Fanuc TP program (LS listing): qwerty_12.ls

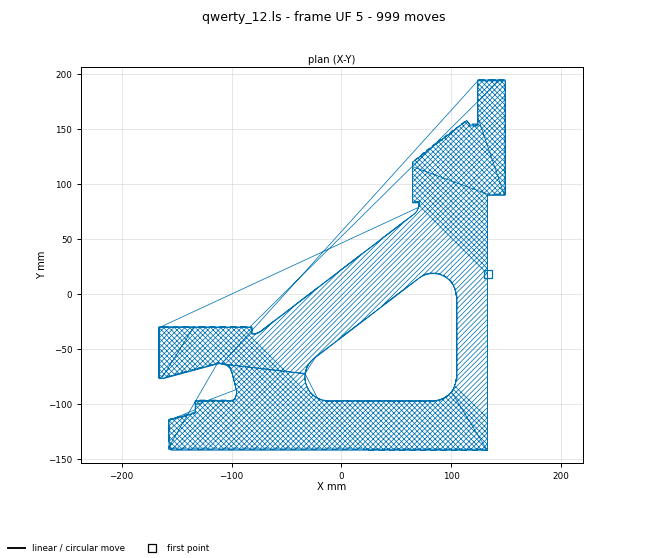
[picture p0: tool path of qwerty_12.ls in frame UF 5, 999 of 999 moves have a stored position in this frame; points joined in program order, loops and branches not executed]
/PROG qwerty_12
/ATTR
OWNER       = MNEDITOR;
CREATE      = DATE 100-11-20  TIME 09:43:21;
MODIFIED    = DATE 100-12-05  TIME 05:26:29;
LINE_COUNT = 999;
PROTECT     = READ_WRITE;
TCD:  STACK_SIZE    = 0,
      TASK_PRIORITY = 50,
      TIME_SLICE    = 0,
      BUSY_LAMP_OFF = 0,
      ABORT_REQUEST = 0,
      PAUSE_REQUEST = 0;
DEFAULT_GROUP   = 1,1,*,*,*;
CONTROL_CODE    = 00000000 00000000;
/MN
1: L P[1] WELD_SPEED CNT100 COORD PTH  ;
2: L P[2] WELD_SPEED CNT100 COORD PTH  ;
3: L P[3] WELD_SPEED CNT100 COORD PTH  ;
4: L P[4] WELD_SPEED CNT100 COORD PTH  ;
5: L P[5] WELD_SPEED CNT100 COORD PTH  ;
6: L P[6] WELD_SPEED CNT100 COORD PTH  ;
7: L P[7] WELD_SPEED CNT100 COORD PTH  ;
8: L P[8] WELD_SPEED CNT100 COORD PTH  ;
9: L P[9] WELD_SPEED CNT100 COORD PTH  ;
10: L P[10] WELD_SPEED CNT100 COORD PTH  ;
11: L P[11] WELD_SPEED CNT100 COORD PTH  ;
12: L P[12] WELD_SPEED CNT100 COORD PTH  ;
13: L P[13] WELD_SPEED CNT100 COORD PTH  ;
14: L P[14] WELD_SPEED CNT100 COORD PTH  ;
15: L P[15] WELD_SPEED CNT100 COORD PTH  ;
16: L P[16] WELD_SPEED CNT100 COORD PTH  ;
17: L P[17] WELD_SPEED CNT100 COORD PTH  ;
18: L P[18] WELD_SPEED CNT100 COORD PTH  ;
19: L P[19] WELD_SPEED CNT100 COORD PTH  ;
20: L P[20] WELD_SPEED CNT100 COORD PTH  ;
21: L P[21] WELD_SPEED CNT100 COORD PTH  ;
22: L P[22] WELD_SPEED CNT100 COORD PTH  ;
23: L P[23] WELD_SPEED CNT100 COORD PTH  ;
24: L P[24] WELD_SPEED CNT100 COORD PTH  ;
25: L P[25] WELD_SPEED CNT100 COORD PTH  ;
26: L P[26] WELD_SPEED CNT100 COORD PTH  ;
27: L P[27] WELD_SPEED CNT100 COORD PTH  ;
28: L P[28] WELD_SPEED CNT100 COORD PTH  ;
29: L P[29] WELD_SPEED CNT100 COORD PTH  ;
30: L P[30] WELD_SPEED CNT100 COORD PTH  ;
31: L P[31] WELD_SPEED CNT100 COORD PTH  ;
32: L P[32] WELD_SPEED CNT100 COORD PTH  ;
33: L P[33] WELD_SPEED CNT100 COORD PTH  ;
34: L P[34] WELD_SPEED CNT100 COORD PTH  ;
35: L P[35] WELD_SPEED CNT100 COORD PTH  ;
36: L P[36] WELD_SPEED CNT100 COORD PTH  ;
37: L P[37] WELD_SPEED CNT100 COORD PTH  ;
38: L P[38] WELD_SPEED CNT100 COORD PTH  ;
39: L P[39] WELD_SPEED CNT100 COORD PTH  ;
40: L P[40] WELD_SPEED CNT100 COORD PTH  ;
41: L P[41] WELD_SPEED CNT100 COORD PTH  ;
42: L P[42] WELD_SPEED CNT100 COORD PTH  ;
43: L P[43] WELD_SPEED CNT100 COORD PTH  ;
44: L P[44] WELD_SPEED CNT100 COORD PTH  ;
45: L P[45] WELD_SPEED CNT100 COORD PTH  ;
46: L P[46] WELD_SPEED CNT100 COORD PTH  ;
47: L P[47] WELD_SPEED CNT100 COORD PTH  ;
48: L P[48] WELD_SPEED CNT100 COORD PTH  ;
49: L P[49] WELD_SPEED CNT100 COORD PTH  ;
50: L P[50] WELD_SPEED CNT100 COORD PTH  ;
51: L P[51] WELD_SPEED CNT100 COORD PTH  ;
52: L P[52] WELD_SPEED CNT100 COORD PTH  ;
53: L P[53] WELD_SPEED CNT100 COORD PTH  ;
54: L P[54] WELD_SPEED CNT100 COORD PTH  ;
55: L P[55] WELD_SPEED CNT100 COORD PTH  ;
56: L P[56] WELD_SPEED CNT100 COORD PTH  ;
57: L P[57] WELD_SPEED CNT100 COORD PTH  ;
58: L P[58] WELD_SPEED CNT100 COORD PTH  ;
59: L P[59] WELD_SPEED CNT100 COORD PTH  ;
60: L P[60] WELD_SPEED CNT100 COORD PTH  ;
61: L P[61] WELD_SPEED CNT100 COORD PTH  ;
62: L P[62] WELD_SPEED CNT100 COORD PTH  ;
63: L P[63] WELD_SPEED CNT100 COORD PTH  ;
64: L P[64] WELD_SPEED CNT100 COORD PTH  ;
65: L P[65] WELD_SPEED CNT100 COORD PTH  ;
66: L P[66] WELD_SPEED CNT100 COORD PTH  ;
67: L P[67] WELD_SPEED CNT100 COORD PTH  ;
68: L P[68] WELD_SPEED CNT100 COORD PTH  ;
69: L P[69] WELD_SPEED CNT100 COORD PTH  ;
70: L P[70] WELD_SPEED CNT100 COORD PTH  ;
71: L P[71] WELD_SPEED CNT100 COORD PTH  ;
72: L P[72] WELD_SPEED CNT100 COORD PTH  ;
73: L P[73] WELD_SPEED CNT100 COORD PTH  ;
74: L P[74] WELD_SPEED CNT100 COORD PTH  ;
75: L P[75] WELD_SPEED CNT100 COORD PTH  ;
76: L P[76] WELD_SPEED CNT100 COORD PTH  ;
77: L P[77] WELD_SPEED CNT100 COORD PTH  ;
78: L P[78] WELD_SPEED CNT100 COORD PTH  ;
79: L P[79] WELD_SPEED CNT100 COORD PTH  ;
80: L P[80] WELD_SPEED CNT100 COORD PTH  ;
81: L P[81] WELD_SPEED CNT100 COORD PTH  ;
82: L P[82] WELD_SPEED CNT100 COORD PTH  ;
83: L P[83] WELD_SPEED CNT100 COORD PTH  ;
84: L P[84] WELD_SPEED CNT100 COORD PTH  ;
85: L P[85] WELD_SPEED CNT100 COORD PTH  ;
86: L P[86] WELD_SPEED CNT100 COORD PTH  ;
87: L P[87] WELD_SPEED CNT100 COORD PTH  ;
88: L P[88] WELD_SPEED CNT100 COORD PTH  ;
: Arc End[1];
89: L P[89] 240cm/min CNT100 COORD  ;
: Arc Start[1];
90: L P[90] WELD_SPEED CNT100 COORD PTH  ;
91: L P[91] WELD_SPEED CNT100 COORD PTH  ;
92: L P[92] WELD_SPEED CNT100 COORD PTH  ;
93: L P[93] WELD_SPEED CNT100 COORD PTH  ;
94: L P[94] WELD_SPEED CNT100 COORD PTH  ;
95: L P[95] WELD_SPEED CNT100 COORD PTH  ;
96: L P[96] WELD_SPEED CNT100 COORD PTH  ;
97: L P[97] WELD_SPEED CNT100 COORD PTH  ;
98: L P[98] WELD_SPEED CNT100 COORD PTH  ;
99: L P[99] WELD_SPEED CNT100 COORD PTH  ;
100: L P[100] WELD_SPEED CNT100 COORD PTH  ;
101: L P[101] WELD_SPEED CNT100 COORD PTH  ;
102: L P[102] WELD_SPEED CNT100 COORD PTH  ;
103: L P[103] WELD_SPEED CNT100 COORD PTH  ;
104: L P[104] WELD_SPEED CNT100 COORD PTH  ;
105: L P[105] WELD_SPEED CNT100 COORD PTH  ;
106: L P[106] WELD_SPEED CNT100 COORD PTH  ;
107: L P[107] WELD_SPEED CNT100 COORD PTH  ;
108: L P[108] WELD_SPEED CNT100 COORD PTH  ;
109: L P[109] WELD_SPEED CNT100 COORD PTH  ;
110: L P[110] WELD_SPEED CNT100 COORD PTH  ;
111: L P[111] WELD_SPEED CNT100 COORD PTH  ;
112: L P[112] WELD_SPEED CNT100 COORD PTH  ;
: Arc End[1];
113: L P[113] 240cm/min CNT100 COORD  ;
: Arc Start[1];
114: L P[114] WELD_SPEED CNT100 COORD PTH  ;
115: L P[115] WELD_SPEED CNT100 COORD PTH  ;
116: L P[116] WELD_SPEED CNT100 COORD PTH  ;
117: L P[117] WELD_SPEED CNT100 COORD PTH  ;
118: L P[118] WELD_SPEED CNT100 COORD PTH  ;
119: L P[119] WELD_SPEED CNT100 COORD PTH  ;
120: L P[120] WELD_SPEED CNT100 COORD PTH  ;
121: L P[121] WELD_SPEED CNT100 COORD PTH  ;
122: L P[122] WELD_SPEED CNT100 COORD PTH  ;
123: L P[123] WELD_SPEED CNT100 COORD PTH  ;
124: L P[124] WELD_SPEED CNT100 COORD PTH  ;
125: L P[125] WELD_SPEED CNT100 COORD PTH  ;
126: L P[126] WELD_SPEED CNT100 COORD PTH  ;
127: L P[127] WELD_SPEED CNT100 COORD PTH  ;
128: L P[128] WELD_SPEED CNT100 COORD PTH  ;
129: L P[129] WELD_SPEED CNT100 COORD PTH  ;
130: L P[130] WELD_SPEED CNT100 COORD PTH  ;
131: L P[131] WELD_SPEED CNT100 COORD PTH  ;
132: L P[132] WELD_SPEED CNT100 COORD PTH  ;
133: L P[133] WELD_SPEED CNT100 COORD PTH  ;
134: L P[134] WELD_SPEED CNT100 COORD PTH  ;
135: L P[135] WELD_SPEED CNT100 COORD PTH  ;
136: L P[136] WELD_SPEED CNT100 COORD PTH  ;
137: L P[137] WELD_SPEED CNT100 COORD PTH  ;
138: L P[138] WELD_SPEED CNT100 COORD PTH  ;
139: L P[139] WELD_SPEED CNT100 COORD PTH  ;
140: L P[140] WELD_SPEED CNT100 COORD PTH  ;
141: L P[141] WELD_SPEED CNT100 COORD PTH  ;
142: L P[142] WELD_SPEED CNT100 COORD PTH  ;
143: L P[143] WELD_SPEED CNT100 COORD PTH  ;
144: L P[144] WELD_SPEED CNT100 COORD PTH  ;
145: L P[145] WELD_SPEED CNT100 COORD PTH  ;
146: L P[146] WELD_SPEED CNT100 COORD PTH  ;
147: L P[147] WELD_SPEED CNT100 COORD PTH  ;
148: L P[148] WELD_SPEED CNT100 COORD PTH  ;
149: L P[149] WELD_SPEED CNT100 COORD PTH  ;
150: L P[150] WELD_SPEED CNT100 COORD PTH  ;
151: L P[151] WELD_SPEED CNT100 COORD PTH  ;
152: L P[152] WELD_SPEED CNT100 COORD PTH  ;
153: L P[153] WELD_SPEED CNT100 COORD PTH  ;
154: L P[154] WELD_SPEED CNT100 COORD PTH  ;
155: L P[155] WELD_SPEED CNT100 COORD PTH  ;
156: L P[156] WELD_SPEED CNT100 COORD PTH  ;
157: L P[157] WELD_SPEED CNT100 COORD PTH  ;
158: L P[158] WELD_SPEED CNT100 COORD PTH  ;
159: L P[159] WELD_SPEED CNT100 COORD PTH  ;
160: L P[160] WELD_SPEED CNT100 COORD PTH  ;
161: L P[161] WELD_SPEED CNT100 COORD PTH  ;
162: L P[162] WELD_SPEED CNT100 COORD PTH  ;
163: L P[163] WELD_SPEED CNT100 COORD PTH  ;
164: L P[164] WELD_SPEED CNT100 COORD PTH  ;
165: L P[165] WELD_SPEED CNT100 COORD PTH  ;
166: L P[166] WELD_SPEED CNT100 COORD PTH  ;
167: L P[167] WELD_SPEED CNT100 COORD PTH  ;
168: L P[168] WELD_SPEED CNT100 COORD PTH  ;
169: L P[169] WELD_SPEED CNT100 COORD PTH  ;
170: L P[170] WELD_SPEED CNT100 COORD PTH  ;
171: L P[171] WELD_SPEED CNT100 COORD PTH  ;
172: L P[172] WELD_SPEED CNT100 COORD PTH  ;
173: L P[173] WELD_SPEED CNT100 COORD PTH  ;
174: L P[174] WELD_SPEED CNT100 COORD PTH  ;
175: L P[175] WELD_SPEED CNT100 COORD PTH  ;
176: L P[176] WELD_SPEED CNT100 COORD PTH  ;
177: L P[177] WELD_SPEED CNT100 COORD PTH  ;
178: L P[178] WELD_SPEED CNT100 COORD PTH  ;
179: L P[179] WELD_SPEED CNT100 COORD PTH  ;
180: L P[180] WELD_SPEED CNT100 COORD PTH  ;
181: L P[181] WELD_SPEED CNT100 COORD PTH  ;
182: L P[182] WELD_SPEED CNT100 COORD PTH  ;
183: L P[183] WELD_SPEED CNT100 COORD PTH  ;
184: L P[184] WELD_SPEED CNT100 COORD PTH  ;
185: L P[185] WELD_SPEED CNT100 COORD PTH  ;
186: L P[186] WELD_SPEED CNT100 COORD PTH  ;
187: L P[187] WELD_SPEED CNT100 COORD PTH  ;
188: L P[188] WELD_SPEED CNT100 COORD PTH  ;
189: L P[189] WELD_SPEED CNT100 COORD PTH  ;
190: L P[190] WELD_SPEED CNT100 COORD PTH  ;
191: L P[191] WELD_SPEED CNT100 COORD PTH  ;
192: L P[192] WELD_SPEED CNT100 COORD PTH  ;
193: L P[193] WELD_SPEED CNT100 COORD PTH  ;
194: L P[194] WELD_SPEED CNT100 COORD PTH  ;
195: L P[195] WELD_SPEED CNT100 COORD PTH  ;
196: L P[196] WELD_SPEED CNT100 COORD PTH  ;
197: L P[197] WELD_SPEED CNT100 COORD PTH  ;
198: L P[198] WELD_SPEED CNT100 COORD PTH  ;
199: L P[199] WELD_SPEED CNT100 COORD PTH  ;
200: L P[200] WELD_SPEED CNT100 COORD PTH  ;
201: L P[201] WELD_SPEED CNT100 COORD PTH  ;
202: L P[202] WELD_SPEED CNT100 COORD PTH  ;
203: L P[203] WELD_SPEED CNT100 COORD PTH  ;
204: L P[204] WELD_SPEED CNT100 COORD PTH  ;
205: L P[205] WELD_SPEED CNT100 COORD PTH  ;
206: L P[206] WELD_SPEED CNT100 COORD PTH  ;
207: L P[207] WELD_SPEED CNT100 COORD PTH  ;
208: L P[208] WELD_SPEED CNT100 COORD PTH  ;
209: L P[209] WELD_SPEED CNT100 COORD PTH  ;
210: L P[210] WELD_SPEED CNT100 COORD PTH  ;
211: L P[211] WELD_SPEED CNT100 COORD PTH  ;
212: L P[212] WELD_SPEED CNT100 COORD PTH  ;
213: L P[213] WELD_SPEED CNT100 COORD PTH  ;
214: L P[214] WELD_SPEED CNT100 COORD PTH  ;
215: L P[215] WELD_SPEED CNT100 COORD PTH  ;
: Arc End[1];
216: L P[216] 240cm/min CNT100 COORD  ;
217: L P[217] 240cm/min CNT100 COORD  ;
: Arc Start[1];
218: L P[218] WELD_SPEED CNT100 COORD PTH  ;
219: L P[219] WELD_SPEED CNT100 COORD PTH  ;
220: L P[220] WELD_SPEED CNT100 COORD PTH  ;
221: L P[221] WELD_SPEED CNT100 COORD PTH  ;
222: L P[222] WELD_SPEED CNT100 COORD PTH  ;
223: L P[223] WELD_SPEED CNT100 COORD PTH  ;
224: L P[224] WELD_SPEED CNT100 COORD PTH  ;
225: L P[225] WELD_SPEED CNT100 COORD PTH  ;
226: L P[226] WELD_SPEED CNT100 COORD PTH  ;
227: L P[227] WELD_SPEED CNT100 COORD PTH  ;
228: L P[228] WELD_SPEED CNT100 COORD PTH  ;
229: L P[229] WELD_SPEED CNT100 COORD PTH  ;
230: L P[230] WELD_SPEED CNT100 COORD PTH  ;
231: L P[231] WELD_SPEED CNT100 COORD PTH  ;
232: L P[232] WELD_SPEED CNT100 COORD PTH  ;
233: L P[233] WELD_SPEED CNT100 COORD PTH  ;
234: L P[234] WELD_SPEED CNT100 COORD PTH  ;
235: L P[235] WELD_SPEED CNT100 COORD PTH  ;
236: L P[236] WELD_SPEED CNT100 COORD PTH  ;
237: L P[237] WELD_SPEED CNT100 COORD PTH  ;
238: L P[238] WELD_SPEED CNT100 COORD PTH  ;
239: L P[239] WELD_SPEED CNT100 COORD PTH  ;
240: L P[240] WELD_SPEED CNT100 COORD PTH  ;
241: L P[241] WELD_SPEED CNT100 COORD PTH  ;
242: L P[242] WELD_SPEED CNT100 COORD PTH  ;
243: L P[243] WELD_SPEED CNT100 COORD PTH  ;
244: L P[244] WELD_SPEED CNT100 COORD PTH  ;
245: L P[245] WELD_SPEED CNT100 COORD PTH  ;
246: L P[246] WELD_SPEED CNT100 COORD PTH  ;
247: L P[247] WELD_SPEED CNT100 COORD PTH  ;
248: L P[248] WELD_SPEED CNT100 COORD PTH  ;
249: L P[249] WELD_SPEED CNT100 COORD PTH  ;
250: L P[250] WELD_SPEED CNT100 COORD PTH  ;
251: L P[251] WELD_SPEED CNT100 COORD PTH  ;
252: L P[252] WELD_SPEED CNT100 COORD PTH  ;
253: L P[253] WELD_SPEED CNT100 COORD PTH  ;
254: L P[254] WELD_SPEED CNT100 COORD PTH  ;
255: L P[255] WELD_SPEED CNT100 COORD PTH  ;
256: L P[256] WELD_SPEED CNT100 COORD PTH  ;
257: L P[257] WELD_SPEED CNT100 COORD PTH  ;
258: L P[258] WELD_SPEED CNT100 COORD PTH  ;
259: L P[259] WELD_SPEED CNT100 COORD PTH  ;
260: L P[260] WELD_SPEED CNT100 COORD PTH  ;
261: L P[261] WELD_SPEED CNT100 COORD PTH  ;
262: L P[262] WELD_SPEED CNT100 COORD PTH  ;
263: L P[263] WELD_SPEED CNT100 COORD PTH  ;
264: L P[264] WELD_SPEED CNT100 COORD PTH  ;
265: L P[265] WELD_SPEED CNT100 COORD PTH  ;
266: L P[266] WELD_SPEED CNT100 COORD PTH  ;
267: L P[267] WELD_SPEED CNT100 COORD PTH  ;
268: L P[268] WELD_SPEED CNT100 COORD PTH  ;
269: L P[269] WELD_SPEED CNT100 COORD PTH  ;
270: L P[270] WELD_SPEED CNT100 COORD PTH  ;
271: L P[271] WELD_SPEED CNT100 COORD PTH  ;
272: L P[272] WELD_SPEED CNT100 COORD PTH  ;
273: L P[273] WELD_SPEED CNT100 COORD PTH  ;
274: L P[274] WELD_SPEED CNT100 COORD PTH  ;
275: L P[275] WELD_SPEED CNT100 COORD PTH  ;
276: L P[276] WELD_SPEED CNT100 COORD PTH  ;
: Arc End[1];
277: L P[277] 240cm/min CNT100 COORD  ;
: Arc Start[1];
278: L P[278] WELD_SPEED CNT100 COORD PTH  ;
279: L P[279] WELD_SPEED CNT100 COORD PTH  ;
280: L P[280] WELD_SPEED CNT100 COORD PTH  ;
281: L P[281] WELD_SPEED CNT100 COORD PTH  ;
282: L P[282] WELD_SPEED CNT100 COORD PTH  ;
283: L P[283] WELD_SPEED CNT100 COORD PTH  ;
284: L P[284] WELD_SPEED CNT100 COORD PTH  ;
285: L P[285] WELD_SPEED CNT100 COORD PTH  ;
286: L P[286] WELD_SPEED CNT100 COORD PTH  ;
287: L P[287] WELD_SPEED CNT100 COORD PTH  ;
288: L P[288] WELD_SPEED CNT100 COORD PTH  ;
289: L P[289] WELD_SPEED CNT100 COORD PTH  ;
290: L P[290] WELD_SPEED CNT100 COORD PTH  ;
291: L P[291] WELD_SPEED CNT100 COORD PTH  ;
292: L P[292] WELD_SPEED CNT100 COORD PTH  ;
293: L P[293] WELD_SPEED CNT100 COORD PTH  ;
294: L P[294] WELD_SPEED CNT100 COORD PTH  ;
295: L P[295] WELD_SPEED CNT100 COORD PTH  ;
296: L P[296] WELD_SPEED CNT100 COORD PTH  ;
297: L P[297] WELD_SPEED CNT100 COORD PTH  ;
298: L P[298] WELD_SPEED CNT100 COORD PTH  ;
299: L P[299] WELD_SPEED CNT100 COORD PTH  ;
300: L P[300] WELD_SPEED CNT100 COORD PTH  ;
301: L P[301] WELD_SPEED CNT100 COORD PTH  ;
302: L P[302] WELD_SPEED CNT100 COORD PTH  ;
303: L P[303] WELD_SPEED CNT100 COORD PTH  ;
304: L P[304] WELD_SPEED CNT100 COORD PTH  ;
305: L P[305] WELD_SPEED CNT100 COORD PTH  ;
306: L P[306] WELD_SPEED CNT100 COORD PTH  ;
307: L P[307] WELD_SPEED CNT100 COORD PTH  ;
308: L P[308] WELD_SPEED CNT100 COORD PTH  ;
309: L P[309] WELD_SPEED CNT100 COORD PTH  ;
310: L P[310] WELD_SPEED CNT100 COORD PTH  ;
311: L P[311] WELD_SPEED CNT100 COORD PTH  ;
312: L P[312] WELD_SPEED CNT100 COORD PTH  ;
313: L P[313] WELD_SPEED CNT100 COORD PTH  ;
314: L P[314] WELD_SPEED CNT100 COORD PTH  ;
315: L P[315] WELD_SPEED CNT100 COORD PTH  ;
316: L P[316] WELD_SPEED CNT100 COORD PTH  ;
317: L P[317] WELD_SPEED CNT100 COORD PTH  ;
318: L P[318] WELD_SPEED CNT100 COORD PTH  ;
319: L P[319] WELD_SPEED CNT100 COORD PTH  ;
320: L P[320] WELD_SPEED CNT100 COORD PTH  ;
321: L P[321] WELD_SPEED CNT100 COORD PTH  ;
322: L P[322] WELD_SPEED CNT100 COORD PTH  ;
323: L P[323] WELD_SPEED CNT100 COORD PTH  ;
324: L P[324] WELD_SPEED CNT100 COORD PTH  ;
325: L P[325] WELD_SPEED CNT100 COORD PTH  ;
326: L P[326] WELD_SPEED CNT100 COORD PTH  ;
327: L P[327] WELD_SPEED CNT100 COORD PTH  ;
328: L P[328] WELD_SPEED CNT100 COORD PTH  ;
329: L P[329] WELD_SPEED CNT100 COORD PTH  ;
330: L P[330] WELD_SPEED CNT100 COORD PTH  ;
331: L P[331] WELD_SPEED CNT100 COORD PTH  ;
332: L P[332] WELD_SPEED CNT100 COORD PTH  ;
333: L P[333] WELD_SPEED CNT100 COORD PTH  ;
334: L P[334] WELD_SPEED CNT100 COORD PTH  ;
335: L P[335] WELD_SPEED CNT100 COORD PTH  ;
336: L P[336] WELD_SPEED CNT100 COORD PTH  ;
337: L P[337] WELD_SPEED CNT100 COORD PTH  ;
338: L P[338] WELD_SPEED CNT100 COORD PTH  ;
339: L P[339] WELD_SPEED CNT100 COORD PTH  ;
340: L P[340] WELD_SPEED CNT100 COORD PTH  ;
341: L P[341] WELD_SPEED CNT100 COORD PTH  ;
342: L P[342] WELD_SPEED CNT100 COORD PTH  ;
343: L P[343] WELD_SPEED CNT100 COORD PTH  ;
344: L P[344] WELD_SPEED CNT100 COORD PTH  ;
345: L P[345] WELD_SPEED CNT100 COORD PTH  ;
346: L P[346] WELD_SPEED CNT100 COORD PTH  ;
347: L P[347] WELD_SPEED CNT100 COORD PTH  ;
348: L P[348] WELD_SPEED CNT100 COORD PTH  ;
349: L P[349] WELD_SPEED CNT100 COORD PTH  ;
350: L P[350] WELD_SPEED CNT100 COORD PTH  ;
351: L P[351] WELD_SPEED CNT100 COORD PTH  ;
352: L P[352] WELD_SPEED CNT100 COORD PTH  ;
353: L P[353] WELD_SPEED CNT100 COORD PTH  ;
354: L P[354] WELD_SPEED CNT100 COORD PTH  ;
355: L P[355] WELD_SPEED CNT100 COORD PTH  ;
356: L P[356] WELD_SPEED CNT100 COORD PTH  ;
357: L P[357] WELD_SPEED CNT100 COORD PTH  ;
358: L P[358] WELD_SPEED CNT100 COORD PTH  ;
359: L P[359] WELD_SPEED CNT100 COORD PTH  ;
360: L P[360] WELD_SPEED CNT100 COORD PTH  ;
361: L P[361] WELD_SPEED CNT100 COORD PTH  ;
362: L P[362] WELD_SPEED CNT100 COORD PTH  ;
363: L P[363] WELD_SPEED CNT100 COORD PTH  ;
364: L P[364] WELD_SPEED CNT100 COORD PTH  ;
365: L P[365] WELD_SPEED CNT100 COORD PTH  ;
366: L P[366] WELD_SPEED CNT100 COORD PTH  ;
367: L P[367] WELD_SPEED CNT100 COORD PTH  ;
368: L P[368] WELD_SPEED CNT100 COORD PTH  ;
369: L P[369] WELD_SPEED CNT100 COORD PTH  ;
370: L P[370] WELD_SPEED CNT100 COORD PTH  ;
371: L P[371] WELD_SPEED CNT100 COORD PTH  ;
372: L P[372] WELD_SPEED CNT100 COORD PTH  ;
373: L P[373] WELD_SPEED CNT100 COORD PTH  ;
374: L P[374] WELD_SPEED CNT100 COORD PTH  ;
375: L P[375] WELD_SPEED CNT100 COORD PTH  ;
376: L P[376] WELD_SPEED CNT100 COORD PTH  ;
377: L P[377] WELD_SPEED CNT100 COORD PTH  ;
378: L P[378] WELD_SPEED CNT100 COORD PTH  ;
379: L P[379] WELD_SPEED CNT100 COORD PTH  ;
380: L P[380] WELD_SPEED CNT100 COORD PTH  ;
381: L P[381] WELD_SPEED CNT100 COORD PTH  ;
382: L P[382] WELD_SPEED CNT100 COORD PTH  ;
383: L P[383] WELD_SPEED CNT100 COORD PTH  ;
384: L P[384] WELD_SPEED CNT100 COORD PTH  ;
385: L P[385] WELD_SPEED CNT100 COORD PTH  ;
386: L P[386] WELD_SPEED CNT100 COORD PTH  ;
387: L P[387] WELD_SPEED CNT100 COORD PTH  ;
: Arc End[1];
388: L P[388] 240cm/min CNT100 COORD  ;
: Arc Start[1];
389: L P[389] WELD_SPEED CNT100 COORD PTH  ;
390: L P[390] WELD_SPEED CNT100 COORD PTH  ;
391: L P[391] WELD_SPEED CNT100 COORD PTH  ;
392: L P[392] WELD_SPEED CNT100 COORD PTH  ;
393: L P[393] WELD_SPEED CNT100 COORD PTH  ;
394: L P[394] WELD_SPEED CNT100 COORD PTH  ;
395: L P[395] WELD_SPEED CNT100 COORD PTH  ;
396: L P[396] WELD_SPEED CNT100 COORD PTH  ;
397: L P[397] WELD_SPEED CNT100 COORD PTH  ;
398: L P[398] WELD_SPEED CNT100 COORD PTH  ;
399: L P[399] WELD_SPEED CNT100 COORD PTH  ;
400: L P[400] WELD_SPEED CNT100 COORD PTH  ;
401: L P[401] WELD_SPEED CNT100 COORD PTH  ;
402: L P[402] WELD_SPEED CNT100 COORD PTH  ;
403: L P[403] WELD_SPEED CNT100 COORD PTH  ;
404: L P[404] WELD_SPEED CNT100 COORD PTH  ;
405: L P[405] WELD_SPEED CNT100 COORD PTH  ;
406: L P[406] WELD_SPEED CNT100 COORD PTH  ;
407: L P[407] WELD_SPEED CNT100 COORD PTH  ;
408: L P[408] WELD_SPEED CNT100 COORD PTH  ;
409: L P[409] WELD_SPEED CNT100 COORD PTH  ;
410: L P[410] WELD_SPEED CNT100 COORD PTH  ;
411: L P[411] WELD_SPEED CNT100 COORD PTH  ;
412: L P[412] WELD_SPEED CNT100 COORD PTH  ;
413: L P[413] WELD_SPEED CNT100 COORD PTH  ;
414: L P[414] WELD_SPEED CNT100 COORD PTH  ;
415: L P[415] WELD_SPEED CNT100 COORD PTH  ;
416: L P[416] WELD_SPEED CNT100 COORD PTH  ;
417: L P[417] WELD_SPEED CNT100 COORD PTH  ;
418: L P[418] WELD_SPEED CNT100 COORD PTH  ;
419: L P[419] WELD_SPEED CNT100 COORD PTH  ;
420: L P[420] WELD_SPEED CNT100 COORD PTH  ;
421: L P[421] WELD_SPEED CNT100 COORD PTH  ;
422: L P[422] WELD_SPEED CNT100 COORD PTH  ;
423: L P[423] WELD_SPEED CNT100 COORD PTH  ;
424: L P[424] WELD_SPEED CNT100 COORD PTH  ;
425: L P[425] WELD_SPEED CNT100 COORD PTH  ;
426: L P[426] WELD_SPEED CNT100 COORD PTH  ;
427: L P[427] WELD_SPEED CNT100 COORD PTH  ;
428: L P[428] WELD_SPEED CNT100 COORD PTH  ;
429: L P[429] WELD_SPEED CNT100 COORD PTH  ;
430: L P[430] WELD_SPEED CNT100 COORD PTH  ;
431: L P[431] WELD_SPEED CNT100 COORD PTH  ;
432: L P[432] WELD_SPEED CNT100 COORD PTH  ;
433: L P[433] WELD_SPEED CNT100 COORD PTH  ;
434: L P[434] WELD_SPEED CNT100 COORD PTH  ;
435: L P[435] WELD_SPEED CNT100 COORD PTH  ;
436: L P[436] WELD_SPEED CNT100 COORD PTH  ;
437: L P[437] WELD_SPEED CNT100 COORD PTH  ;
438: L P[438] WELD_SPEED CNT100 COORD PTH  ;
439: L P[439] WELD_SPEED CNT100 COORD PTH  ;
440: L P[440] WELD_SPEED CNT100 COORD PTH  ;
441: L P[441] WELD_SPEED CNT100 COORD PTH  ;
442: L P[442] WELD_SPEED CNT100 COORD PTH  ;
443: L P[443] WELD_SPEED CNT100 COORD PTH  ;
444: L P[444] WELD_SPEED CNT100 COORD PTH  ;
445: L P[445] WELD_SPEED CNT100 COORD PTH  ;
446: L P[446] WELD_SPEED CNT100 COORD PTH  ;
447: L P[447] WELD_SPEED CNT100 COORD PTH  ;
448: L P[448] WELD_SPEED CNT100 COORD PTH  ;
449: L P[449] WELD_SPEED CNT100 COORD PTH  ;
450: L P[450] WELD_SPEED CNT100 COORD PTH  ;
451: L P[451] WELD_SPEED CNT100 COORD PTH  ;
452: L P[452] WELD_SPEED CNT100 COORD PTH  ;
453: L P[453] WELD_SPEED CNT100 COORD PTH  ;
454: L P[454] WELD_SPEED CNT100 COORD PTH  ;
455: L P[455] WELD_SPEED CNT100 COORD PTH  ;
456: L P[456] WELD_SPEED CNT100 COORD PTH  ;
457: L P[457] WELD_SPEED CNT100 COORD PTH  ;
458: L P[458] WELD_SPEED CNT100 COORD PTH  ;
459: L P[459] WELD_SPEED CNT100 COORD PTH  ;
460: L P[460] WELD_SPEED CNT100 COORD PTH  ;
461: L P[461] WELD_SPEED CNT100 COORD PTH  ;
462: L P[462] WELD_SPEED CNT100 COORD PTH  ;
463: L P[463] WELD_SPEED CNT100 COORD PTH  ;
464: L P[464] WELD_SPEED CNT100 COORD PTH  ;
465: L P[465] WELD_SPEED CNT100 COORD PTH  ;
466: L P[466] WELD_SPEED CNT100 COORD PTH  ;
467: L P[467] WELD_SPEED CNT100 COORD PTH  ;
468: L P[468] WELD_SPEED CNT100 COORD PTH  ;
469: L P[469] WELD_SPEED CNT100 COORD PTH  ;
470: L P[470] WELD_SPEED CNT100 COORD PTH  ;
471: L P[471] WELD_SPEED CNT100 COORD PTH  ;
472: L P[472] WELD_SPEED CNT100 COORD PTH  ;
473: L P[473] WELD_SPEED CNT100 COORD PTH  ;
474: L P[474] WELD_SPEED CNT100 COORD PTH  ;
475: L P[475] WELD_SPEED CNT100 COORD PTH  ;
476: L P[476] WELD_SPEED CNT100 COORD PTH  ;
477: L P[477] WELD_SPEED CNT100 COORD PTH  ;
478: L P[478] WELD_SPEED CNT100 COORD PTH  ;
479: L P[479] WELD_SPEED CNT100 COORD PTH  ;
480: L P[480] WELD_SPEED CNT100 COORD PTH  ;
481: L P[481] WELD_SPEED CNT100 COORD PTH  ;
: Arc End[1];
482: L P[482] 240cm/min CNT100 COORD  ;
: Arc Start[1];
483: L P[483] WELD_SPEED CNT100 COORD PTH  ;
484: L P[484] WELD_SPEED CNT100 COORD PTH  ;
485: L P[485] WELD_SPEED CNT100 COORD PTH  ;
486: L P[486] WELD_SPEED CNT100 COORD PTH  ;
487: L P[487] WELD_SPEED CNT100 COORD PTH  ;
488: L P[488] WELD_SPEED CNT100 COORD PTH  ;
489: L P[489] WELD_SPEED CNT100 COORD PTH  ;
490: L P[490] WELD_SPEED CNT100 COORD PTH  ;
491: L P[491] WELD_SPEED CNT100 COORD PTH  ;
492: L P[492] WELD_SPEED CNT100 COORD PTH  ;
493: L P[493] WELD_SPEED CNT100 COORD PTH  ;
494: L P[494] WELD_SPEED CNT100 COORD PTH  ;
495: L P[495] WELD_SPEED CNT100 COORD PTH  ;
496: L P[496] WELD_SPEED CNT100 COORD PTH  ;
497: L P[497] WELD_SPEED CNT100 COORD PTH  ;
498: L P[498] WELD_SPEED CNT100 COORD PTH  ;
499: L P[499] WELD_SPEED CNT100 COORD PTH  ;
500: L P[500] WELD_SPEED CNT100 COORD PTH  ;
501: L P[501] WELD_SPEED CNT100 COORD PTH  ;
502: L P[502] WELD_SPEED CNT100 COORD PTH  ;
503: L P[503] WELD_SPEED CNT100 COORD PTH  ;
504: L P[504] WELD_SPEED CNT100 COORD PTH  ;
505: L P[505] WELD_SPEED CNT100 COORD PTH  ;
506: L P[506] WELD_SPEED CNT100 COORD PTH  ;
507: L P[507] WELD_SPEED CNT100 COORD PTH  ;
508: L P[508] WELD_SPEED CNT100 COORD PTH  ;
509: L P[509] WELD_SPEED CNT100 COORD PTH  ;
510: L P[510] WELD_SPEED CNT100 COORD PTH  ;
511: L P[511] WELD_SPEED CNT100 COORD PTH  ;
512: L P[512] WELD_SPEED CNT100 COORD PTH  ;
513: L P[513] WELD_SPEED CNT100 COORD PTH  ;
514: L P[514] WELD_SPEED CNT100 COORD PTH  ;
515: L P[515] WELD_SPEED CNT100 COORD PTH  ;
516: L P[516] WELD_SPEED CNT100 COORD PTH  ;
517: L P[517] WELD_SPEED CNT100 COORD PTH  ;
518: L P[518] WELD_SPEED CNT100 COORD PTH  ;
519: L P[519] WELD_SPEED CNT100 COORD PTH  ;
520: L P[520] WELD_SPEED CNT100 COORD PTH  ;
521: L P[521] WELD_SPEED CNT100 COORD PTH  ;
522: L P[522] WELD_SPEED CNT100 COORD PTH  ;
523: L P[523] WELD_SPEED CNT100 COORD PTH  ;
524: L P[524] WELD_SPEED CNT100 COORD PTH  ;
525: L P[525] WELD_SPEED CNT100 COORD PTH  ;
526: L P[526] WELD_SPEED CNT100 COORD PTH  ;
527: L P[527] WELD_SPEED CNT100 COORD PTH  ;
528: L P[528] WELD_SPEED CNT100 COORD PTH  ;
529: L P[529] WELD_SPEED CNT100 COORD PTH  ;
530: L P[530] WELD_SPEED CNT100 COORD PTH  ;
531: L P[531] WELD_SPEED CNT100 COORD PTH  ;
532: L P[532] WELD_SPEED CNT100 COORD PTH  ;
533: L P[533] WELD_SPEED CNT100 COORD PTH  ;
534: L P[534] WELD_SPEED CNT100 COORD PTH  ;
535: L P[535] WELD_SPEED CNT100 COORD PTH  ;
536: L P[536] WELD_SPEED CNT100 COORD PTH  ;
537: L P[537] WELD_SPEED CNT100 COORD PTH  ;
538: L P[538] WELD_SPEED CNT100 COORD PTH  ;
539: L P[539] WELD_SPEED CNT100 COORD PTH  ;
540: L P[540] WELD_SPEED CNT100 COORD PTH  ;
541: L P[541] WELD_SPEED CNT100 COORD PTH  ;
542: L P[542] WELD_SPEED CNT100 COORD PTH  ;
543: L P[543] WELD_SPEED CNT100 COORD PTH  ;
544: L P[544] WELD_SPEED CNT100 COORD PTH  ;
545: L P[545] WELD_SPEED CNT100 COORD PTH  ;
546: L P[546] WELD_SPEED CNT100 COORD PTH  ;
547: L P[547] WELD_SPEED CNT100 COORD PTH  ;
548: L P[548] WELD_SPEED CNT100 COORD PTH  ;
549: L P[549] WELD_SPEED CNT100 COORD PTH  ;
550: L P[550] WELD_SPEED CNT100 COORD PTH  ;
551: L P[551] WELD_SPEED CNT100 COORD PTH  ;
552: L P[552] WELD_SPEED CNT100 COORD PTH  ;
553: L P[553] WELD_SPEED CNT100 COORD PTH  ;
554: L P[554] WELD_SPEED CNT100 COORD PTH  ;
555: L P[555] WELD_SPEED CNT100 COORD PTH  ;
556: L P[556] WELD_SPEED CNT100 COORD PTH  ;
557: L P[557] WELD_SPEED CNT100 COORD PTH  ;
558: L P[558] WELD_SPEED CNT100 COORD PTH  ;
559: L P[559] WELD_SPEED CNT100 COORD PTH  ;
560: L P[560] WELD_SPEED CNT100 COORD PTH  ;
561: L P[561] WELD_SPEED CNT100 COORD PTH  ;
562: L P[562] WELD_SPEED CNT100 COORD PTH  ;
563: L P[563] WELD_SPEED CNT100 COORD PTH  ;
564: L P[564] WELD_SPEED CNT100 COORD PTH  ;
565: L P[565] WELD_SPEED CNT100 COORD PTH  ;
566: L P[566] WELD_SPEED CNT100 COORD PTH  ;
567: L P[567] WELD_SPEED CNT100 COORD PTH  ;
568: L P[568] WELD_SPEED CNT100 COORD PTH  ;
569: L P[569] WELD_SPEED CNT100 COORD PTH  ;
570: L P[570] WELD_SPEED CNT100 COORD PTH  ;
571: L P[571] WELD_SPEED CNT100 COORD PTH  ;
572: L P[572] WELD_SPEED CNT100 COORD PTH  ;
573: L P[573] WELD_SPEED CNT100 COORD PTH  ;
574: L P[574] WELD_SPEED CNT100 COORD PTH  ;
575: L P[575] WELD_SPEED CNT100 COORD PTH  ;
576: L P[576] WELD_SPEED CNT100 COORD PTH  ;
577: L P[577] WELD_SPEED CNT100 COORD PTH  ;
578: L P[578] WELD_SPEED CNT100 COORD PTH  ;
579: L P[579] WELD_SPEED CNT100 COORD PTH  ;
580: L P[580] WELD_SPEED CNT100 COORD PTH  ;
581: L P[581] WELD_SPEED CNT100 COORD PTH  ;
582: L P[582] WELD_SPEED CNT100 COORD PTH  ;
583: L P[583] WELD_SPEED CNT100 COORD PTH  ;
584: L P[584] WELD_SPEED CNT100 COORD PTH  ;
585: L P[585] WELD_SPEED CNT100 COORD PTH  ;
586: L P[586] WELD_SPEED CNT100 COORD PTH  ;
587: L P[587] WELD_SPEED CNT100 COORD PTH  ;
588: L P[588] WELD_SPEED CNT100 COORD PTH  ;
589: L P[589] WELD_SPEED CNT100 COORD PTH  ;
590: L P[590] WELD_SPEED CNT100 COORD PTH  ;
591: L P[591] WELD_SPEED CNT100 COORD PTH  ;
592: L P[592] WELD_SPEED CNT100 COORD PTH  ;
593: L P[593] WELD_SPEED CNT100 COORD PTH  ;
594: L P[594] WELD_SPEED CNT100 COORD PTH  ;
595: L P[595] WELD_SPEED CNT100 COORD PTH  ;
596: L P[596] WELD_SPEED CNT100 COORD PTH  ;
597: L P[597] WELD_SPEED CNT100 COORD PTH  ;
598: L P[598] WELD_SPEED CNT100 COORD PTH  ;
599: L P[599] WELD_SPEED CNT100 COORD PTH  ;
600: L P[600] WELD_SPEED CNT100 COORD PTH  ;
601: L P[601] WELD_SPEED CNT100 COORD PTH  ;
602: L P[602] WELD_SPEED CNT100 COORD PTH  ;
603: L P[603] WELD_SPEED CNT100 COORD PTH  ;
604: L P[604] WELD_SPEED CNT100 COORD PTH  ;
605: L P[605] WELD_SPEED CNT100 COORD PTH  ;
606: L P[606] WELD_SPEED CNT100 COORD PTH  ;
607: L P[607] WELD_SPEED CNT100 COORD PTH  ;
608: L P[608] WELD_SPEED CNT100 COORD PTH  ;
609: L P[609] WELD_SPEED CNT100 COORD PTH  ;
610: L P[610] WELD_SPEED CNT100 COORD PTH  ;
611: L P[611] WELD_SPEED CNT100 COORD PTH  ;
612: L P[612] WELD_SPEED CNT100 COORD PTH  ;
613: L P[613] WELD_SPEED CNT100 COORD PTH  ;
614: L P[614] WELD_SPEED CNT100 COORD PTH  ;
615: L P[615] WELD_SPEED CNT100 COORD PTH  ;
616: L P[616] WELD_SPEED CNT100 COORD PTH  ;
617: L P[617] WELD_SPEED CNT100 COORD PTH  ;
618: L P[618] WELD_SPEED CNT100 COORD PTH  ;
619: L P[619] WELD_SPEED CNT100 COORD PTH  ;
620: L P[620] WELD_SPEED CNT100 COORD PTH  ;
621: L P[621] WELD_SPEED CNT100 COORD PTH  ;
622: L P[622] WELD_SPEED CNT100 COORD PTH  ;
623: L P[623] WELD_SPEED CNT100 COORD PTH  ;
624: L P[624] WELD_SPEED CNT100 COORD PTH  ;
625: L P[625] WELD_SPEED CNT100 COORD PTH  ;
626: L P[626] WELD_SPEED CNT100 COORD PTH  ;
627: L P[627] WELD_SPEED CNT100 COORD PTH  ;
628: L P[628] WELD_SPEED CNT100 COORD PTH  ;
629: L P[629] WELD_SPEED CNT100 COORD PTH  ;
630: L P[630] WELD_SPEED CNT100 COORD PTH  ;
631: L P[631] WELD_SPEED CNT100 COORD PTH  ;
632: L P[632] WELD_SPEED CNT100 COORD PTH  ;
633: L P[633] WELD_SPEED CNT100 COORD PTH  ;
634: L P[634] WELD_SPEED CNT100 COORD PTH  ;
635: L P[635] WELD_SPEED CNT100 COORD PTH  ;
636: L P[636] WELD_SPEED CNT100 COORD PTH  ;
637: L P[637] WELD_SPEED CNT100 COORD PTH  ;
638: L P[638] WELD_SPEED CNT100 COORD PTH  ;
639: L P[639] WELD_SPEED CNT100 COORD PTH  ;
640: L P[640] WELD_SPEED CNT100 COORD PTH  ;
641: L P[641] WELD_SPEED CNT100 COORD PTH  ;
642: L P[642] WELD_SPEED CNT100 COORD PTH  ;
643: L P[643] WELD_SPEED CNT100 COORD PTH  ;
644: L P[644] WELD_SPEED CNT100 COORD PTH  ;
645: L P[645] WELD_SPEED CNT100 COORD PTH  ;
646: L P[646] WELD_SPEED CNT100 COORD PTH  ;
647: L P[647] WELD_SPEED CNT100 COORD PTH  ;
648: L P[648] WELD_SPEED CNT100 COORD PTH  ;
649: L P[649] WELD_SPEED CNT100 COORD PTH  ;
650: L P[650] WELD_SPEED CNT100 COORD PTH  ;
: Arc End[1];
651: L P[651] 240cm/min CNT100 COORD  ;
: Arc Start[1];
652: L P[652] WELD_SPEED CNT100 COORD PTH  ;
653: L P[653] WELD_SPEED CNT100 COORD PTH  ;
654: L P[654] WELD_SPEED CNT100 COORD PTH  ;
: Arc End[1];
655: L P[655] 240cm/min CNT100 COORD  ;
: Arc Start[1];
656: L P[656] WELD_SPEED CNT100 COORD PTH  ;
657: L P[657] WELD_SPEED CNT100 COORD PTH  ;
658: L P[658] WELD_SPEED CNT100 COORD PTH  ;
659: L P[659] WELD_SPEED CNT100 COORD PTH  ;
660: L P[660] WELD_SPEED CNT100 COORD PTH  ;
661: L P[661] WELD_SPEED CNT100 COORD PTH  ;
662: L P[662] WELD_SPEED CNT100 COORD PTH  ;
663: L P[663] WELD_SPEED CNT100 COORD PTH  ;
664: L P[664] WELD_SPEED CNT100 COORD PTH  ;
665: L P[665] WELD_SPEED CNT100 COORD PTH  ;
666: L P[666] WELD_SPEED CNT100 COORD PTH  ;
667: L P[667] WELD_SPEED CNT100 COORD PTH  ;
668: L P[668] WELD_SPEED CNT100 COORD PTH  ;
669: L P[669] WELD_SPEED CNT100 COORD PTH  ;
670: L P[670] WELD_SPEED CNT100 COORD PTH  ;
671: L P[671] WELD_SPEED CNT100 COORD PTH  ;
672: L P[672] WELD_SPEED CNT100 COORD PTH  ;
673: L P[673] WELD_SPEED CNT100 COORD PTH  ;
674: L P[674] WELD_SPEED CNT100 COORD PTH  ;
675: L P[675] WELD_SPEED CNT100 COORD PTH  ;
676: L P[676] WELD_SPEED CNT100 COORD PTH  ;
677: L P[677] WELD_SPEED CNT100 COORD PTH  ;
678: L P[678] WELD_SPEED CNT100 COORD PTH  ;
679: L P[679] WELD_SPEED CNT100 COORD PTH  ;
680: L P[680] WELD_SPEED CNT100 COORD PTH  ;
681: L P[681] WELD_SPEED CNT100 COORD PTH  ;
682: L P[682] WELD_SPEED CNT100 COORD PTH  ;
683: L P[683] WELD_SPEED CNT100 COORD PTH  ;
684: L P[684] WELD_SPEED CNT100 COORD PTH  ;
685: L P[685] WELD_SPEED CNT100 COORD PTH  ;
686: L P[686] WELD_SPEED CNT100 COORD PTH  ;
687: L P[687] WELD_SPEED CNT100 COORD PTH  ;
688: L P[688] WELD_SPEED CNT100 COORD PTH  ;
689: L P[689] WELD_SPEED CNT100 COORD PTH  ;
690: L P[690] WELD_SPEED CNT100 COORD PTH  ;
691: L P[691] WELD_SPEED CNT100 COORD PTH  ;
692: L P[692] WELD_SPEED CNT100 COORD PTH  ;
693: L P[693] WELD_SPEED CNT100 COORD PTH  ;
694: L P[694] WELD_SPEED CNT100 COORD PTH  ;
695: L P[695] WELD_SPEED CNT100 COORD PTH  ;
696: L P[696] WELD_SPEED CNT100 COORD PTH  ;
697: L P[697] WELD_SPEED CNT100 COORD PTH  ;
698: L P[698] WELD_SPEED CNT100 COORD PTH  ;
699: L P[699] WELD_SPEED CNT100 COORD PTH  ;
700: L P[700] WELD_SPEED CNT100 COORD PTH  ;
701: L P[701] WELD_SPEED CNT100 COORD PTH  ;
702: L P[702] WELD_SPEED CNT100 COORD PTH  ;
703: L P[703] WELD_SPEED CNT100 COORD PTH  ;
704: L P[704] WELD_SPEED CNT100 COORD PTH  ;
705: L P[705] WELD_SPEED CNT100 COORD PTH  ;
706: L P[706] WELD_SPEED CNT100 COORD PTH  ;
707: L P[707] WELD_SPEED CNT100 COORD PTH  ;
708: L P[708] WELD_SPEED CNT100 COORD PTH  ;
709: L P[709] WELD_SPEED CNT100 COORD PTH  ;
710: L P[710] WELD_SPEED CNT100 COORD PTH  ;
711: L P[711] WELD_SPEED CNT100 COORD PTH  ;
712: L P[712] WELD_SPEED CNT100 COORD PTH  ;
713: L P[713] WELD_SPEED CNT100 COORD PTH  ;
714: L P[714] WELD_SPEED CNT100 COORD PTH  ;
715: L P[715] WELD_SPEED CNT100 COORD PTH  ;
716: L P[716] WELD_SPEED CNT100 COORD PTH  ;
717: L P[717] WELD_SPEED CNT100 COORD PTH  ;
718: L P[718] WELD_SPEED CNT100 COORD PTH  ;
719: L P[719] WELD_SPEED CNT100 COORD PTH  ;
: Arc End[1];
720: L P[720] 240cm/min CNT100 COORD  ;
: Arc Start[1];
721: L P[721] WELD_SPEED CNT100 COORD PTH  ;
722: L P[722] WELD_SPEED CNT100 COORD PTH  ;
723: L P[723] WELD_SPEED CNT100 COORD PTH  ;
724: L P[724] WELD_SPEED CNT100 COORD PTH  ;
725: L P[725] WELD_SPEED CNT100 COORD PTH  ;
726: L P[726] WELD_SPEED CNT100 COORD PTH  ;
727: L P[727] WELD_SPEED CNT100 COORD PTH  ;
728: L P[728] WELD_SPEED CNT100 COORD PTH  ;
729: L P[729] WELD_SPEED CNT100 COORD PTH  ;
730: L P[730] WELD_SPEED CNT100 COORD PTH  ;
731: L P[731] WELD_SPEED CNT100 COORD PTH  ;
732: L P[732] WELD_SPEED CNT100 COORD PTH  ;
733: L P[733] WELD_SPEED CNT100 COORD PTH  ;
734: L P[734] WELD_SPEED CNT100 COORD PTH  ;
735: L P[735] WELD_SPEED CNT100 COORD PTH  ;
736: L P[736] WELD_SPEED CNT100 COORD PTH  ;
737: L P[737] WELD_SPEED CNT100 COORD PTH  ;
738: L P[738] WELD_SPEED CNT100 COORD PTH  ;
739: L P[739] WELD_SPEED CNT100 COORD PTH  ;
740: L P[740] WELD_SPEED CNT100 COORD PTH  ;
741: L P[741] WELD_SPEED CNT100 COORD PTH  ;
742: L P[742] WELD_SPEED CNT100 COORD PTH  ;
: Arc End[1];
743: L P[743] 240cm/min CNT100 COORD  ;
: Arc Start[1];
744: L P[744] WELD_SPEED CNT100 COORD PTH  ;
745: L P[745] WELD_SPEED CNT100 COORD PTH  ;
746: L P[746] WELD_SPEED CNT100 COORD PTH  ;
747: L P[747] WELD_SPEED CNT100 COORD PTH  ;
748: L P[748] WELD_SPEED CNT100 COORD PTH  ;
749: L P[749] WELD_SPEED CNT100 COORD PTH  ;
750: L P[750] WELD_SPEED CNT100 COORD PTH  ;
: Arc End[1];
751: L P[751] 240cm/min CNT100 COORD  ;
: Arc Start[1];
752: L P[752] WELD_SPEED CNT100 COORD PTH  ;
753: L P[753] WELD_SPEED CNT100 COORD PTH  ;
754: L P[754] WELD_SPEED CNT100 COORD PTH  ;
755: L P[755] WELD_SPEED CNT100 COORD PTH  ;
756: L P[756] WELD_SPEED CNT100 COORD PTH  ;
757: L P[757] WELD_SPEED CNT100 COORD PTH  ;
758: L P[758] WELD_SPEED CNT100 COORD PTH  ;
759: L P[759] WELD_SPEED CNT100 COORD PTH  ;
760: L P[760] WELD_SPEED CNT100 COORD PTH  ;
761: L P[761] WELD_SPEED CNT100 COORD PTH  ;
762: L P[762] WELD_SPEED CNT100 COORD PTH  ;
763: L P[763] WELD_SPEED CNT100 COORD PTH  ;
764: L P[764] WELD_SPEED CNT100 COORD PTH  ;
765: L P[765] WELD_SPEED CNT100 COORD PTH  ;
766: L P[766] WELD_SPEED CNT100 COORD PTH  ;
: Arc End[1];
767: L P[767] 240cm/min CNT100 COORD  ;
768: L P[768] 240cm/min CNT100 COORD  ;
: Arc Start[1];
769: L P[769] WELD_SPEED CNT100 COORD PTH  ;
770: L P[770] WELD_SPEED CNT100 COORD PTH  ;
771: L P[771] WELD_SPEED CNT100 COORD PTH  ;
772: L P[772] WELD_SPEED CNT100 COORD PTH  ;
773: L P[773] WELD_SPEED CNT100 COORD PTH  ;
774: L P[774] WELD_SPEED CNT100 COORD PTH  ;
775: L P[775] WELD_SPEED CNT100 COORD PTH  ;
776: L P[776] WELD_SPEED CNT100 COORD PTH  ;
777: L P[777] WELD_SPEED CNT100 COORD PTH  ;
778: L P[778] WELD_SPEED CNT100 COORD PTH  ;
779: L P[779] WELD_SPEED CNT100 COORD PTH  ;
780: L P[780] WELD_SPEED CNT100 COORD PTH  ;
781: L P[781] WELD_SPEED CNT100 COORD PTH  ;
782: L P[782] WELD_SPEED CNT100 COORD PTH  ;
783: L P[783] WELD_SPEED CNT100 COORD PTH  ;
784: L P[784] WELD_SPEED CNT100 COORD PTH  ;
785: L P[785] WELD_SPEED CNT100 COORD PTH  ;
786: L P[786] WELD_SPEED CNT100 COORD PTH  ;
787: L P[787] WELD_SPEED CNT100 COORD PTH  ;
788: L P[788] WELD_SPEED CNT100 COORD PTH  ;
789: L P[789] WELD_SPEED CNT100 COORD PTH  ;
790: L P[790] WELD_SPEED CNT100 COORD PTH  ;
791: L P[791] WELD_SPEED CNT100 COORD PTH  ;
792: L P[792] WELD_SPEED CNT100 COORD PTH  ;
793: L P[793] WELD_SPEED CNT100 COORD PTH  ;
794: L P[794] WELD_SPEED CNT100 COORD PTH  ;
795: L P[795] WELD_SPEED CNT100 COORD PTH  ;
796: L P[796] WELD_SPEED CNT100 COORD PTH  ;
797: L P[797] WELD_SPEED CNT100 COORD PTH  ;
798: L P[798] WELD_SPEED CNT100 COORD PTH  ;
799: L P[799] WELD_SPEED CNT100 COORD PTH  ;
800: L P[800] WELD_SPEED CNT100 COORD PTH  ;
801: L P[801] WELD_SPEED CNT100 COORD PTH  ;
802: L P[802] WELD_SPEED CNT100 COORD PTH  ;
803: L P[803] WELD_SPEED CNT100 COORD PTH  ;
804: L P[804] WELD_SPEED CNT100 COORD PTH  ;
805: L P[805] WELD_SPEED CNT100 COORD PTH  ;
806: L P[806] WELD_SPEED CNT100 COORD PTH  ;
807: L P[807] WELD_SPEED CNT100 COORD PTH  ;
808: L P[808] WELD_SPEED CNT100 COORD PTH  ;
809: L P[809] WELD_SPEED CNT100 COORD PTH  ;
810: L P[810] WELD_SPEED CNT100 COORD PTH  ;
811: L P[811] WELD_SPEED CNT100 COORD PTH  ;
812: L P[812] WELD_SPEED CNT100 COORD PTH  ;
813: L P[813] WELD_SPEED CNT100 COORD PTH  ;
814: L P[814] WELD_SPEED CNT100 COORD PTH  ;
815: L P[815] WELD_SPEED CNT100 COORD PTH  ;
816: L P[816] WELD_SPEED CNT100 COORD PTH  ;
817: L P[817] WELD_SPEED CNT100 COORD PTH  ;
818: L P[818] WELD_SPEED CNT100 COORD PTH  ;
819: L P[819] WELD_SPEED CNT100 COORD PTH  ;
820: L P[820] WELD_SPEED CNT100 COORD PTH  ;
821: L P[821] WELD_SPEED CNT100 COORD PTH  ;
822: L P[822] WELD_SPEED CNT100 COORD PTH  ;
823: L P[823] WELD_SPEED CNT100 COORD PTH  ;
824: L P[824] WELD_SPEED CNT100 COORD PTH  ;
825: L P[825] WELD_SPEED CNT100 COORD PTH  ;
826: L P[826] WELD_SPEED CNT100 COORD PTH  ;
827: L P[827] WELD_SPEED CNT100 COORD PTH  ;
828: L P[828] WELD_SPEED CNT100 COORD PTH  ;
: Arc End[1];
829: L P[829] 240cm/min CNT100 COORD  ;
: Arc Start[1];
830: L P[830] WELD_SPEED CNT100 COORD PTH  ;
831: L P[831] WELD_SPEED CNT100 COORD PTH  ;
832: L P[832] WELD_SPEED CNT100 COORD PTH  ;
833: L P[833] WELD_SPEED CNT100 COORD PTH  ;
834: L P[834] WELD_SPEED CNT100 COORD PTH  ;
835: L P[835] WELD_SPEED CNT100 COORD PTH  ;
836: L P[836] WELD_SPEED CNT100 COORD PTH  ;
837: L P[837] WELD_SPEED CNT100 COORD PTH  ;
838: L P[838] WELD_SPEED CNT100 COORD PTH  ;
839: L P[839] WELD_SPEED CNT100 COORD PTH  ;
840: L P[840] WELD_SPEED CNT100 COORD PTH  ;
841: L P[841] WELD_SPEED CNT100 COORD PTH  ;
842: L P[842] WELD_SPEED CNT100 COORD PTH  ;
843: L P[843] WELD_SPEED CNT100 COORD PTH  ;
844: L P[844] WELD_SPEED CNT100 COORD PTH  ;
845: L P[845] WELD_SPEED CNT100 COORD PTH  ;
846: L P[846] WELD_SPEED CNT100 COORD PTH  ;
847: L P[847] WELD_SPEED CNT100 COORD PTH  ;
848: L P[848] WELD_SPEED CNT100 COORD PTH  ;
849: L P[849] WELD_SPEED CNT100 COORD PTH  ;
850: L P[850] WELD_SPEED CNT100 COORD PTH  ;
851: L P[851] WELD_SPEED CNT100 COORD PTH  ;
852: L P[852] WELD_SPEED CNT100 COORD PTH  ;
853: L P[853] WELD_SPEED CNT100 COORD PTH  ;
854: L P[854] WELD_SPEED CNT100 COORD PTH  ;
855: L P[855] WELD_SPEED CNT100 COORD PTH  ;
856: L P[856] WELD_SPEED CNT100 COORD PTH  ;
857: L P[857] WELD_SPEED CNT100 COORD PTH  ;
858: L P[858] WELD_SPEED CNT100 COORD PTH  ;
859: L P[859] WELD_SPEED CNT100 COORD PTH  ;
860: L P[860] WELD_SPEED CNT100 COORD PTH  ;
861: L P[861] WELD_SPEED CNT100 COORD PTH  ;
862: L P[862] WELD_SPEED CNT100 COORD PTH  ;
863: L P[863] WELD_SPEED CNT100 COORD PTH  ;
864: L P[864] WELD_SPEED CNT100 COORD PTH  ;
865: L P[865] WELD_SPEED CNT100 COORD PTH  ;
866: L P[866] WELD_SPEED CNT100 COORD PTH  ;
867: L P[867] WELD_SPEED CNT100 COORD PTH  ;
868: L P[868] WELD_SPEED CNT100 COORD PTH  ;
869: L P[869] WELD_SPEED CNT100 COORD PTH  ;
870: L P[870] WELD_SPEED CNT100 COORD PTH  ;
871: L P[871] WELD_SPEED CNT100 COORD PTH  ;
872: L P[872] WELD_SPEED CNT100 COORD PTH  ;
873: L P[873] WELD_SPEED CNT100 COORD PTH  ;
874: L P[874] WELD_SPEED CNT100 COORD PTH  ;
875: L P[875] WELD_SPEED CNT100 COORD PTH  ;
876: L P[876] WELD_SPEED CNT100 COORD PTH  ;
877: L P[877] WELD_SPEED CNT100 COORD PTH  ;
878: L P[878] WELD_SPEED CNT100 COORD PTH  ;
879: L P[879] WELD_SPEED CNT100 COORD PTH  ;
880: L P[880] WELD_SPEED CNT100 COORD PTH  ;
881: L P[881] WELD_SPEED CNT100 COORD PTH  ;
882: L P[882] WELD_SPEED CNT100 COORD PTH  ;
883: L P[883] WELD_SPEED CNT100 COORD PTH  ;
884: L P[884] WELD_SPEED CNT100 COORD PTH  ;
885: L P[885] WELD_SPEED CNT100 COORD PTH  ;
886: L P[886] WELD_SPEED CNT100 COORD PTH  ;
887: L P[887] WELD_SPEED CNT100 COORD PTH  ;
888: L P[888] WELD_SPEED CNT100 COORD PTH  ;
889: L P[889] WELD_SPEED CNT100 COORD PTH  ;
890: L P[890] WELD_SPEED CNT100 COORD PTH  ;
891: L P[891] WELD_SPEED CNT100 COORD PTH  ;
892: L P[892] WELD_SPEED CNT100 COORD PTH  ;
893: L P[893] WELD_SPEED CNT100 COORD PTH  ;
894: L P[894] WELD_SPEED CNT100 COORD PTH  ;
895: L P[895] WELD_SPEED CNT100 COORD PTH  ;
896: L P[896] WELD_SPEED CNT100 COORD PTH  ;
897: L P[897] WELD_SPEED CNT100 COORD PTH  ;
898: L P[898] WELD_SPEED CNT100 COORD PTH  ;
899: L P[899] WELD_SPEED CNT100 COORD PTH  ;
900: L P[900] WELD_SPEED CNT100 COORD PTH  ;
901: L P[901] WELD_SPEED CNT100 COORD PTH  ;
902: L P[902] WELD_SPEED CNT100 COORD PTH  ;
903: L P[903] WELD_SPEED CNT100 COORD PTH  ;
904: L P[904] WELD_SPEED CNT100 COORD PTH  ;
905: L P[905] WELD_SPEED CNT100 COORD PTH  ;
906: L P[906] WELD_SPEED CNT100 COORD PTH  ;
907: L P[907] WELD_SPEED CNT100 COORD PTH  ;
908: L P[908] WELD_SPEED CNT100 COORD PTH  ;
909: L P[909] WELD_SPEED CNT100 COORD PTH  ;
910: L P[910] WELD_SPEED CNT100 COORD PTH  ;
911: L P[911] WELD_SPEED CNT100 COORD PTH  ;
912: L P[912] WELD_SPEED CNT100 COORD PTH  ;
913: L P[913] WELD_SPEED CNT100 COORD PTH  ;
914: L P[914] WELD_SPEED CNT100 COORD PTH  ;
915: L P[915] WELD_SPEED CNT100 COORD PTH  ;
916: L P[916] WELD_SPEED CNT100 COORD PTH  ;
917: L P[917] WELD_SPEED CNT100 COORD PTH  ;
918: L P[918] WELD_SPEED CNT100 COORD PTH  ;
919: L P[919] WELD_SPEED CNT100 COORD PTH  ;
920: L P[920] WELD_SPEED CNT100 COORD PTH  ;
921: L P[921] WELD_SPEED CNT100 COORD PTH  ;
922: L P[922] WELD_SPEED CNT100 COORD PTH  ;
923: L P[923] WELD_SPEED CNT100 COORD PTH  ;
924: L P[924] WELD_SPEED CNT100 COORD PTH  ;
925: L P[925] WELD_SPEED CNT100 COORD PTH  ;
926: L P[926] WELD_SPEED CNT100 COORD PTH  ;
927: L P[927] WELD_SPEED CNT100 COORD PTH  ;
: Arc End[1];
928: L P[928] 240cm/min CNT100 COORD  ;
: Arc Start[1];
929: L P[929] WELD_SPEED CNT100 COORD PTH  ;
930: L P[930] WELD_SPEED CNT100 COORD PTH  ;
931: L P[931] WELD_SPEED CNT100 COORD PTH  ;
932: L P[932] WELD_SPEED CNT100 COORD PTH  ;
933: L P[933] WELD_SPEED CNT100 COORD PTH  ;
934: L P[934] WELD_SPEED CNT100 COORD PTH  ;
935: L P[935] WELD_SPEED CNT100 COORD PTH  ;
936: L P[936] WELD_SPEED CNT100 COORD PTH  ;
937: L P[937] WELD_SPEED CNT100 COORD PTH  ;
938: L P[938] WELD_SPEED CNT100 COORD PTH  ;
939: L P[939] WELD_SPEED CNT100 COORD PTH  ;
940: L P[940] WELD_SPEED CNT100 COORD PTH  ;
941: L P[941] WELD_SPEED CNT100 COORD PTH  ;
942: L P[942] WELD_SPEED CNT100 COORD PTH  ;
943: L P[943] WELD_SPEED CNT100 COORD PTH  ;
944: L P[944] WELD_SPEED CNT100 COORD PTH  ;
945: L P[945] WELD_SPEED CNT100 COORD PTH  ;
946: L P[946] WELD_SPEED CNT100 COORD PTH  ;
947: L P[947] WELD_SPEED CNT100 COORD PTH  ;
948: L P[948] WELD_SPEED CNT100 COORD PTH  ;
949: L P[949] WELD_SPEED CNT100 COORD PTH  ;
950: L P[950] WELD_SPEED CNT100 COORD PTH  ;
951: L P[951] WELD_SPEED CNT100 COORD PTH  ;
952: L P[952] WELD_SPEED CNT100 COORD PTH  ;
953: L P[953] WELD_SPEED CNT100 COORD PTH  ;
954: L P[954] WELD_SPEED CNT100 COORD PTH  ;
955: L P[955] WELD_SPEED CNT100 COORD PTH  ;
956: L P[956] WELD_SPEED CNT100 COORD PTH  ;
957: L P[957] WELD_SPEED CNT100 COORD PTH  ;
958: L P[958] WELD_SPEED CNT100 COORD PTH  ;
959: L P[959] WELD_SPEED CNT100 COORD PTH  ;
960: L P[960] WELD_SPEED CNT100 COORD PTH  ;
961: L P[961] WELD_SPEED CNT100 COORD PTH  ;
962: L P[962] WELD_SPEED CNT100 COORD PTH  ;
963: L P[963] WELD_SPEED CNT100 COORD PTH  ;
964: L P[964] WELD_SPEED CNT100 COORD PTH  ;
965: L P[965] WELD_SPEED CNT100 COORD PTH  ;
966: L P[966] WELD_SPEED CNT100 COORD PTH  ;
967: L P[967] WELD_SPEED CNT100 COORD PTH  ;
968: L P[968] WELD_SPEED CNT100 COORD PTH  ;
969: L P[969] WELD_SPEED CNT100 COORD PTH  ;
970: L P[970] WELD_SPEED CNT100 COORD PTH  ;
971: L P[971] WELD_SPEED CNT100 COORD PTH  ;
972: L P[972] WELD_SPEED CNT100 COORD PTH  ;
973: L P[973] WELD_SPEED CNT100 COORD PTH  ;
974: L P[974] WELD_SPEED CNT100 COORD PTH  ;
975: L P[975] WELD_SPEED CNT100 COORD PTH  ;
976: L P[976] WELD_SPEED CNT100 COORD PTH  ;
977: L P[977] WELD_SPEED CNT100 COORD PTH  ;
978: L P[978] WELD_SPEED CNT100 COORD PTH  ;
979: L P[979] WELD_SPEED CNT100 COORD PTH  ;
980: L P[980] WELD_SPEED CNT100 COORD PTH  ;
981: L P[981] WELD_SPEED CNT100 COORD PTH  ;
982: L P[982] WELD_SPEED CNT100 COORD PTH  ;
983: L P[983] WELD_SPEED CNT100 COORD PTH  ;
984: L P[984] WELD_SPEED CNT100 COORD PTH  ;
985: L P[985] WELD_SPEED CNT100 COORD PTH  ;
986: L P[986] WELD_SPEED CNT100 COORD PTH  ;
987: L P[987] WELD_SPEED CNT100 COORD PTH  ;
988: L P[988] WELD_SPEED CNT100 COORD PTH  ;
989: L P[989] WELD_SPEED CNT100 COORD PTH  ;
990: L P[990] WELD_SPEED CNT100 COORD PTH  ;
991: L P[991] WELD_SPEED CNT100 COORD PTH  ;
992: L P[992] WELD_SPEED CNT100 COORD PTH  ;
993: L P[993] WELD_SPEED CNT100 COORD PTH  ;
994: L P[994] WELD_SPEED CNT100 COORD PTH  ;
995: L P[995] WELD_SPEED CNT100 COORD PTH  ;
996: L P[996] WELD_SPEED CNT100 COORD PTH  ;
997: L P[997] WELD_SPEED CNT100 COORD PTH  ;
998: L P[998] WELD_SPEED CNT100 COORD PTH  ;
999: L P[999] WELD_SPEED CNT100 COORD PTH  ;
: CALL qwerty_13;
/POS
P[1] {
   GP1:
       UF : 5, UT : 6,     CONFIG: 'N U T, 0, 0, 0',
      X = 133.0 mm, Y = 18.4 mm, Z = 85.8 mm,
      W = 0.0 deg, P = 0.0 deg, R = 0.0 deg
   GP2:
       UF : 1, UT : 2,
      J1 = 0.0 deg, J2 = 0.0 deg
};
P[2] {
   GP1:
       UF : 5, UT : 6,     CONFIG: 'N U T, 0, 0, 0',
      X = 70.5 mm, Y = 80.9 mm, Z = 85.8 mm,
      W = 0.0 deg, P = 0.0 deg, R = 0.0 deg
   GP2:
       UF : 1, UT : 2,
      J1 = 0.0 deg, J2 = 0.0 deg
};
P[3] {
   GP1:
       UF : 5, UT : 6,     CONFIG: 'N U T, 0, 0, 0',
      X = 70.6 mm, Y = 81.6 mm, Z = 85.8 mm,
      W = 0.0 deg, P = 0.0 deg, R = 0.0 deg
   GP2:
       UF : 1, UT : 2,
      J1 = 0.0 deg, J2 = 0.0 deg
};
P[4] {
   GP1:
       UF : 5, UT : 6,     CONFIG: 'N U T, 0, 0, 0',
      X = 70.8 mm, Y = 84.2 mm, Z = 85.8 mm,
      W = 0.0 deg, P = 0.0 deg, R = 0.0 deg
   GP2:
       UF : 1, UT : 2,
      J1 = 0.0 deg, J2 = 0.0 deg
};
P[5] {
   GP1:
       UF : 5, UT : 6,     CONFIG: 'N U T, 0, 0, 0',
      X = 67.1 mm, Y = 84.2 mm, Z = 85.8 mm,
      W = 0.0 deg, P = 0.0 deg, R = 0.0 deg
   GP2:
       UF : 1, UT : 2,
      J1 = 0.0 deg, J2 = 0.0 deg
};
P[6] {
   GP1:
       UF : 5, UT : 6,     CONFIG: 'N U T, 0, 0, 0',
      X = 64.7 mm, Y = 86.7 mm, Z = 85.8 mm,
      W = 0.0 deg, P = 0.0 deg, R = 0.0 deg
   GP2:
       UF : 1, UT : 2,
      J1 = 0.0 deg, J2 = 0.0 deg
};
P[7] {
   GP1:
       UF : 5, UT : 6,     CONFIG: 'N U T, 0, 0, 0',
      X = 64.7 mm, Y = 91.4 mm, Z = 85.8 mm,
      W = 0.0 deg, P = 0.0 deg, R = 0.0 deg
   GP2:
       UF : 1, UT : 2,
      J1 = 0.0 deg, J2 = 0.0 deg
};
P[8] {
   GP1:
       UF : 5, UT : 6,     CONFIG: 'N U T, 0, 0, 0',
      X = 133.0 mm, Y = 23.1 mm, Z = 85.8 mm,
      W = 0.0 deg, P = 0.0 deg, R = 0.0 deg
   GP2:
       UF : 1, UT : 2,
      J1 = 0.0 deg, J2 = 0.0 deg
};
P[9] {
   GP1:
       UF : 5, UT : 6,     CONFIG: 'N U T, 0, 0, 0',
      X = 133.0 mm, Y = 27.8 mm, Z = 85.8 mm,
      W = 0.0 deg, P = 0.0 deg, R = 0.0 deg
   GP2:
       UF : 1, UT : 2,
      J1 = 0.0 deg, J2 = 0.0 deg
};
P[10] {
   GP1:
       UF : 5, UT : 6,     CONFIG: 'N U T, 0, 0, 0',
      X = 64.7 mm, Y = 96.1 mm, Z = 85.8 mm,
      W = 0.0 deg, P = 0.0 deg, R = 0.0 deg
   GP2:
       UF : 1, UT : 2,
      J1 = 0.0 deg, J2 = 0.0 deg
};
P[11] {
   GP1:
       UF : 5, UT : 6,     CONFIG: 'N U T, 0, 0, 0',
      X = 64.7 mm, Y = 101.0 mm, Z = 85.8 mm,
      W = 0.0 deg, P = 0.0 deg, R = 0.0 deg
   GP2:
       UF : 1, UT : 2,
      J1 = 0.0 deg, J2 = 0.0 deg
};
P[12] {
   GP1:
       UF : 5, UT : 6,     CONFIG: 'N U T, 0, 0, 0',
      X = 133.0 mm, Y = 32.5 mm, Z = 85.8 mm,
      W = 0.0 deg, P = 0.0 deg, R = 0.0 deg
   GP2:
       UF : 1, UT : 2,
      J1 = 0.0 deg, J2 = 0.0 deg
};
P[13] {
   GP1:
       UF : 5, UT : 6,     CONFIG: 'N U T, 0, 0, 0',
      X = 133.0 mm, Y = 37.2 mm, Z = 85.8 mm,
      W = 0.0 deg, P = 0.0 deg, R = 0.0 deg
   GP2:
       UF : 1, UT : 2,
      J1 = 0.0 deg, J2 = 0.0 deg
};
P[14] {
   GP1:
       UF : 5, UT : 6,     CONFIG: 'N U T, 0, 0, 0',
      X = 64.7 mm, Y = 106.0 mm, Z = 85.8 mm,
      W = 0.0 deg, P = 0.0 deg, R = 0.0 deg
   GP2:
       UF : 1, UT : 2,
      J1 = 0.0 deg, J2 = 0.0 deg
};
P[15] {
   GP1:
       UF : 5, UT : 6,     CONFIG: 'N U T, 0, 0, 0',
      X = 64.7 mm, Y = 110.0 mm, Z = 85.8 mm,
      W = 0.0 deg, P = 0.0 deg, R = 0.0 deg
   GP2:
       UF : 1, UT : 2,
      J1 = 0.0 deg, J2 = 0.0 deg
};
P[16] {
   GP1:
       UF : 5, UT : 6,     CONFIG: 'N U T, 0, 0, 0',
      X = 133.0 mm, Y = 41.9 mm, Z = 85.8 mm,
      W = 0.0 deg, P = 0.0 deg, R = 0.0 deg
   GP2:
       UF : 1, UT : 2,
      J1 = 0.0 deg, J2 = 0.0 deg
};
P[17] {
   GP1:
       UF : 5, UT : 6,     CONFIG: 'N U T, 0, 0, 0',
      X = 133.0 mm, Y = 46.6 mm, Z = 85.8 mm,
      W = 0.0 deg, P = 0.0 deg, R = 0.0 deg
   GP2:
       UF : 1, UT : 2,
      J1 = 0.0 deg, J2 = 0.0 deg
};
P[18] {
   GP1:
       UF : 5, UT : 6,     CONFIG: 'N U T, 0, 0, 0',
      X = 64.7 mm, Y = 115.0 mm, Z = 85.8 mm,
      W = 0.0 deg, P = 0.0 deg, R = 0.0 deg
   GP2:
       UF : 1, UT : 2,
      J1 = 0.0 deg, J2 = 0.0 deg
};
P[19] {
   GP1:
       UF : 5, UT : 6,     CONFIG: 'N U T, 0, 0, 0',
      X = 64.7 mm, Y = 120.0 mm, Z = 85.8 mm,
      W = 0.0 deg, P = 0.0 deg, R = 0.0 deg
   GP2:
       UF : 1, UT : 2,
      J1 = 0.0 deg, J2 = 0.0 deg
};
P[20] {
   GP1:
       UF : 5, UT : 6,     CONFIG: 'N U T, 0, 0, 0',
      X = 133.0 mm, Y = 51.3 mm, Z = 85.8 mm,
      W = 0.0 deg, P = 0.0 deg, R = 0.0 deg
   GP2:
       UF : 1, UT : 2,
      J1 = 0.0 deg, J2 = 0.0 deg
};
P[21] {
   GP1:
       UF : 5, UT : 6,     CONFIG: 'N U T, 0, 0, 0',
      X = 133.0 mm, Y = 56.0 mm, Z = 85.8 mm,
      W = 0.0 deg, P = 0.0 deg, R = 0.0 deg
   GP2:
       UF : 1, UT : 2,
      J1 = 0.0 deg, J2 = 0.0 deg
};
P[22] {
   GP1:
       UF : 5, UT : 6,     CONFIG: 'N U T, 0, 0, 0',
      X = 66.6 mm, Y = 122.0 mm, Z = 85.8 mm,
      W = 0.0 deg, P = 0.0 deg, R = 0.0 deg
   GP2:
       UF : 1, UT : 2,
      J1 = 0.0 deg, J2 = 0.0 deg
};
P[23] {
   GP1:
       UF : 5, UT : 6,     CONFIG: 'N U T, 0, 0, 0',
      X = 69.3 mm, Y = 124.0 mm, Z = 85.8 mm,
      W = 0.0 deg, P = 0.0 deg, R = 0.0 deg
   GP2:
       UF : 1, UT : 2,
      J1 = 0.0 deg, J2 = 0.0 deg
};
P[24] {
   GP1:
       UF : 5, UT : 6,     CONFIG: 'N U T, 0, 0, 0',
      X = 133.0 mm, Y = 60.7 mm, Z = 85.8 mm,
      W = 0.0 deg, P = 0.0 deg, R = 0.0 deg
   GP2:
       UF : 1, UT : 2,
      J1 = 0.0 deg, J2 = 0.0 deg
};
P[25] {
   GP1:
       UF : 5, UT : 6,     CONFIG: 'N U T, 0, 0, 0',
      X = 133.0 mm, Y = 65.4 mm, Z = 85.8 mm,
      W = 0.0 deg, P = 0.0 deg, R = 0.0 deg
   GP2:
       UF : 1, UT : 2,
      J1 = 0.0 deg, J2 = 0.0 deg
};
P[26] {
   GP1:
       UF : 5, UT : 6,     CONFIG: 'N U T, 0, 0, 0',
      X = 71.9 mm, Y = 126.0 mm, Z = 85.8 mm,
      W = 0.0 deg, P = 0.0 deg, R = 0.0 deg
   GP2:
       UF : 1, UT : 2,
      J1 = 0.0 deg, J2 = 0.0 deg
};
P[27] {
   GP1:
       UF : 5, UT : 6,     CONFIG: 'N U T, 0, 0, 0',
      X = 74.6 mm, Y = 129.0 mm, Z = 85.8 mm,
      W = 0.0 deg, P = 0.0 deg, R = 0.0 deg
   GP2:
       UF : 1, UT : 2,
      J1 = 0.0 deg, J2 = 0.0 deg
};
P[28] {
   GP1:
       UF : 5, UT : 6,     CONFIG: 'N U T, 0, 0, 0',
      X = 133.0 mm, Y = 70.1 mm, Z = 85.8 mm,
      W = 0.0 deg, P = 0.0 deg, R = 0.0 deg
   GP2:
       UF : 1, UT : 2,
      J1 = 0.0 deg, J2 = 0.0 deg
};
P[29] {
   GP1:
       UF : 5, UT : 6,     CONFIG: 'N U T, 0, 0, 0',
      X = 133.0 mm, Y = 74.8 mm, Z = 85.8 mm,
      W = 0.0 deg, P = 0.0 deg, R = 0.0 deg
   GP2:
       UF : 1, UT : 2,
      J1 = 0.0 deg, J2 = 0.0 deg
};
P[30] {
   GP1:
       UF : 5, UT : 6,     CONFIG: 'N U T, 0, 0, 0',
      X = 77.3 mm, Y = 131.0 mm, Z = 85.8 mm,
      W = 0.0 deg, P = 0.0 deg, R = 0.0 deg
   GP2:
       UF : 1, UT : 2,
      J1 = 0.0 deg, J2 = 0.0 deg
};
P[31] {
   GP1:
       UF : 5, UT : 6,     CONFIG: 'N U T, 0, 0, 0',
      X = 79.9 mm, Y = 133.0 mm, Z = 85.8 mm,
      W = 0.0 deg, P = 0.0 deg, R = 0.0 deg
   GP2:
       UF : 1, UT : 2,
      J1 = 0.0 deg, J2 = 0.0 deg
};
P[32] {
   GP1:
       UF : 5, UT : 6,     CONFIG: 'N U T, 0, 0, 0',
      X = 133.0 mm, Y = 79.5 mm, Z = 85.8 mm,
      W = 0.0 deg, P = 0.0 deg, R = 0.0 deg
   GP2:
       UF : 1, UT : 2,
      J1 = 0.0 deg, J2 = 0.0 deg
};
P[33] {
   GP1:
       UF : 5, UT : 6,     CONFIG: 'N U T, 0, 0, 0',
      X = 133.0 mm, Y = 84.2 mm, Z = 85.8 mm,
      W = 0.0 deg, P = 0.0 deg, R = 0.0 deg
   GP2:
       UF : 1, UT : 2,
      J1 = 0.0 deg, J2 = 0.0 deg
};
P[34] {
   GP1:
       UF : 5, UT : 6,     CONFIG: 'N U T, 0, 0, 0',
      X = 82.6 mm, Y = 135.0 mm, Z = 85.8 mm,
      W = 0.0 deg, P = 0.0 deg, R = 0.0 deg
   GP2:
       UF : 1, UT : 2,
      J1 = 0.0 deg, J2 = 0.0 deg
};
P[35] {
   GP1:
       UF : 5, UT : 6,     CONFIG: 'N U T, 0, 0, 0',
      X = 85.3 mm, Y = 137.0 mm, Z = 85.8 mm,
      W = 0.0 deg, P = 0.0 deg, R = 0.0 deg
   GP2:
       UF : 1, UT : 2,
      J1 = 0.0 deg, J2 = 0.0 deg
};
P[36] {
   GP1:
       UF : 5, UT : 6,     CONFIG: 'N U T, 0, 0, 0',
      X = 133.0 mm, Y = 88.9 mm, Z = 85.8 mm,
      W = 0.0 deg, P = 0.0 deg, R = 0.0 deg
   GP2:
       UF : 1, UT : 2,
      J1 = 0.0 deg, J2 = 0.0 deg
};
P[37] {
   GP1:
       UF : 5, UT : 6,     CONFIG: 'N U T, 0, 0, 0',
      X = 133.0 mm, Y = 91.2 mm, Z = 85.8 mm,
      W = 0.0 deg, P = 0.0 deg, R = 0.0 deg
   GP2:
       UF : 1, UT : 2,
      J1 = 0.0 deg, J2 = 0.0 deg
};
P[38] {
   GP1:
       UF : 5, UT : 6,     CONFIG: 'N U T, 0, 0, 0',
      X = 135.0 mm, Y = 91.2 mm, Z = 85.8 mm,
      W = 0.0 deg, P = 0.0 deg, R = 0.0 deg
   GP2:
       UF : 1, UT : 2,
      J1 = 0.0 deg, J2 = 0.0 deg
};
P[39] {
   GP1:
       UF : 5, UT : 6,     CONFIG: 'N U T, 0, 0, 0',
      X = 87.9 mm, Y = 139.0 mm, Z = 85.8 mm,
      W = 0.0 deg, P = 0.0 deg, R = 0.0 deg
   GP2:
       UF : 1, UT : 2,
      J1 = 0.0 deg, J2 = 0.0 deg
};
P[40] {
   GP1:
       UF : 5, UT : 6,     CONFIG: 'N U T, 0, 0, 0',
      X = 90.6 mm, Y = 141.0 mm, Z = 85.8 mm,
      W = 0.0 deg, P = 0.0 deg, R = 0.0 deg
   GP2:
       UF : 1, UT : 2,
      J1 = 0.0 deg, J2 = 0.0 deg
};
P[41] {
   GP1:
       UF : 5, UT : 6,     CONFIG: 'N U T, 0, 0, 0',
      X = 140.0 mm, Y = 91.2 mm, Z = 85.8 mm,
      W = 0.0 deg, P = 0.0 deg, R = 0.0 deg
   GP2:
       UF : 1, UT : 2,
      J1 = 0.0 deg, J2 = 0.0 deg
};
P[42] {
   GP1:
       UF : 5, UT : 6,     CONFIG: 'N U T, 0, 0, 0',
      X = 145.0 mm, Y = 91.2 mm, Z = 85.8 mm,
      W = 0.0 deg, P = 0.0 deg, R = 0.0 deg
   GP2:
       UF : 1, UT : 2,
      J1 = 0.0 deg, J2 = 0.0 deg
};
P[43] {
   GP1:
       UF : 5, UT : 6,     CONFIG: 'N U T, 0, 0, 0',
      X = 93.2 mm, Y = 143.0 mm, Z = 85.8 mm,
      W = 0.0 deg, P = 0.0 deg, R = 0.0 deg
   GP2:
       UF : 1, UT : 2,
      J1 = 0.0 deg, J2 = 0.0 deg
};
P[44] {
   GP1:
       UF : 5, UT : 6,     CONFIG: 'N U T, 0, 0, 0',
      X = 95.9 mm, Y = 145.0 mm, Z = 85.8 mm,
      W = 0.0 deg, P = 0.0 deg, R = 0.0 deg
   GP2:
       UF : 1, UT : 2,
      J1 = 0.0 deg, J2 = 0.0 deg
};
P[45] {
   GP1:
       UF : 5, UT : 6,     CONFIG: 'N U T, 0, 0, 0',
      X = 149.0 mm, Y = 91.7 mm, Z = 85.8 mm,
      W = 0.0 deg, P = 0.0 deg, R = 0.0 deg
   GP2:
       UF : 1, UT : 2,
      J1 = 0.0 deg, J2 = 0.0 deg
};
P[46] {
   GP1:
       UF : 5, UT : 6,     CONFIG: 'N U T, 0, 0, 0',
      X = 149.0 mm, Y = 96.4 mm, Z = 85.8 mm,
      W = 0.0 deg, P = 0.0 deg, R = 0.0 deg
   GP2:
       UF : 1, UT : 2,
      J1 = 0.0 deg, J2 = 0.0 deg
};
P[47] {
   GP1:
       UF : 5, UT : 6,     CONFIG: 'N U T, 0, 0, 0',
      X = 98.6 mm, Y = 147.0 mm, Z = 85.8 mm,
      W = 0.0 deg, P = 0.0 deg, R = 0.0 deg
   GP2:
       UF : 1, UT : 2,
      J1 = 0.0 deg, J2 = 0.0 deg
};
P[48] {
   GP1:
       UF : 5, UT : 6,     CONFIG: 'N U T, 0, 0, 0',
      X = 101.0 mm, Y = 149.0 mm, Z = 85.8 mm,
      W = 0.0 deg, P = 0.0 deg, R = 0.0 deg
   GP2:
       UF : 1, UT : 2,
      J1 = 0.0 deg, J2 = 0.0 deg
};
P[49] {
   GP1:
       UF : 5, UT : 6,     CONFIG: 'N U T, 0, 0, 0',
      X = 149.0 mm, Y = 101.0 mm, Z = 85.8 mm,
      W = 0.0 deg, P = 0.0 deg, R = 0.0 deg
   GP2:
       UF : 1, UT : 2,
      J1 = 0.0 deg, J2 = 0.0 deg
};
P[50] {
   GP1:
       UF : 5, UT : 6,     CONFIG: 'N U T, 0, 0, 0',
      X = 149.0 mm, Y = 106.0 mm, Z = 85.8 mm,
      W = 0.0 deg, P = 0.0 deg, R = 0.0 deg
   GP2:
       UF : 1, UT : 2,
      J1 = 0.0 deg, J2 = 0.0 deg
};
P[51] {
   GP1:
       UF : 5, UT : 6,     CONFIG: 'N U T, 0, 0, 0',
      X = 104.0 mm, Y = 151.0 mm, Z = 85.8 mm,
      W = 0.0 deg, P = 0.0 deg, R = 0.0 deg
   GP2:
       UF : 1, UT : 2,
      J1 = 0.0 deg, J2 = 0.0 deg
};
P[52] {
   GP1:
       UF : 5, UT : 6,     CONFIG: 'N U T, 0, 0, 0',
      X = 107.0 mm, Y = 153.0 mm, Z = 85.8 mm,
      W = 0.0 deg, P = 0.0 deg, R = 0.0 deg
   GP2:
       UF : 1, UT : 2,
      J1 = 0.0 deg, J2 = 0.0 deg
};
P[53] {
   GP1:
       UF : 5, UT : 6,     CONFIG: 'N U T, 0, 0, 0',
      X = 149.0 mm, Y = 111.0 mm, Z = 85.8 mm,
      W = 0.0 deg, P = 0.0 deg, R = 0.0 deg
   GP2:
       UF : 1, UT : 2,
      J1 = 0.0 deg, J2 = 0.0 deg
};
P[54] {
   GP1:
       UF : 5, UT : 6,     CONFIG: 'N U T, 0, 0, 0',
      X = 149.0 mm, Y = 115.0 mm, Z = 85.8 mm,
      W = 0.0 deg, P = 0.0 deg, R = 0.0 deg
   GP2:
       UF : 1, UT : 2,
      J1 = 0.0 deg, J2 = 0.0 deg
};
P[55] {
   GP1:
       UF : 5, UT : 6,     CONFIG: 'N U T, 0, 0, 0',
      X = 109.0 mm, Y = 155.0 mm, Z = 85.8 mm,
      W = 0.0 deg, P = 0.0 deg, R = 0.0 deg
   GP2:
       UF : 1, UT : 2,
      J1 = 0.0 deg, J2 = 0.0 deg
};
P[56] {
   GP1:
       UF : 5, UT : 6,     CONFIG: 'N U T, 0, 0, 0',
      X = 112.0 mm, Y = 157.0 mm, Z = 85.8 mm,
      W = 0.0 deg, P = 0.0 deg, R = 0.0 deg
   GP2:
       UF : 1, UT : 2,
      J1 = 0.0 deg, J2 = 0.0 deg
};
P[57] {
   GP1:
       UF : 5, UT : 6,     CONFIG: 'N U T, 0, 0, 0',
      X = 149.0 mm, Y = 120.0 mm, Z = 85.8 mm,
      W = 0.0 deg, P = 0.0 deg, R = 0.0 deg
   GP2:
       UF : 1, UT : 2,
      J1 = 0.0 deg, J2 = 0.0 deg
};
P[58] {
   GP1:
       UF : 5, UT : 6,     CONFIG: 'N U T, 0, 0, 0',
      X = 149.0 mm, Y = 125.0 mm, Z = 85.8 mm,
      W = 0.0 deg, P = 0.0 deg, R = 0.0 deg
   GP2:
       UF : 1, UT : 2,
      J1 = 0.0 deg, J2 = 0.0 deg
};
P[59] {
   GP1:
       UF : 5, UT : 6,     CONFIG: 'N U T, 0, 0, 0',
      X = 119.0 mm, Y = 155.0 mm, Z = 85.8 mm,
      W = 0.0 deg, P = 0.0 deg, R = 0.0 deg
   GP2:
       UF : 1, UT : 2,
      J1 = 0.0 deg, J2 = 0.0 deg
};
P[60] {
   GP1:
       UF : 5, UT : 6,     CONFIG: 'N U T, 0, 0, 0',
      X = 124.0 mm, Y = 155.0 mm, Z = 85.8 mm,
      W = 0.0 deg, P = 0.0 deg, R = 0.0 deg
   GP2:
       UF : 1, UT : 2,
      J1 = 0.0 deg, J2 = 0.0 deg
};
P[61] {
   GP1:
       UF : 5, UT : 6,     CONFIG: 'N U T, 0, 0, 0',
      X = 124.0 mm, Y = 155.0 mm, Z = 85.8 mm,
      W = 0.0 deg, P = 0.0 deg, R = 0.0 deg
   GP2:
       UF : 1, UT : 2,
      J1 = 0.0 deg, J2 = 0.0 deg
};
P[62] {
   GP1:
       UF : 5, UT : 6,     CONFIG: 'N U T, 0, 0, 0',
      X = 149.0 mm, Y = 129.0 mm, Z = 85.8 mm,
      W = 0.0 deg, P = 0.0 deg, R = 0.0 deg
   GP2:
       UF : 1, UT : 2,
      J1 = 0.0 deg, J2 = 0.0 deg
};
P[63] {
   GP1:
       UF : 5, UT : 6,     CONFIG: 'N U T, 0, 0, 0',
      X = 149.0 mm, Y = 134.0 mm, Z = 85.8 mm,
      W = 0.0 deg, P = 0.0 deg, R = 0.0 deg
   GP2:
       UF : 1, UT : 2,
      J1 = 0.0 deg, J2 = 0.0 deg
};
P[64] {
   GP1:
       UF : 5, UT : 6,     CONFIG: 'N U T, 0, 0, 0',
      X = 124.0 mm, Y = 159.0 mm, Z = 85.8 mm,
      W = 0.0 deg, P = 0.0 deg, R = 0.0 deg
   GP2:
       UF : 1, UT : 2,
      J1 = 0.0 deg, J2 = 0.0 deg
};
P[65] {
   GP1:
       UF : 5, UT : 6,     CONFIG: 'N U T, 0, 0, 0',
      X = 124.0 mm, Y = 164.0 mm, Z = 85.8 mm,
      W = 0.0 deg, P = 0.0 deg, R = 0.0 deg
   GP2:
       UF : 1, UT : 2,
      J1 = 0.0 deg, J2 = 0.0 deg
};
P[66] {
   GP1:
       UF : 5, UT : 6,     CONFIG: 'N U T, 0, 0, 0',
      X = 149.0 mm, Y = 139.0 mm, Z = 85.8 mm,
      W = 0.0 deg, P = 0.0 deg, R = 0.0 deg
   GP2:
       UF : 1, UT : 2,
      J1 = 0.0 deg, J2 = 0.0 deg
};
P[67] {
   GP1:
       UF : 5, UT : 6,     CONFIG: 'N U T, 0, 0, 0',
      X = 149.0 mm, Y = 143.0 mm, Z = 85.8 mm,
      W = 0.0 deg, P = 0.0 deg, R = 0.0 deg
   GP2:
       UF : 1, UT : 2,
      J1 = 0.0 deg, J2 = 0.0 deg
};
P[68] {
   GP1:
       UF : 5, UT : 6,     CONFIG: 'N U T, 0, 0, 0',
      X = 124.0 mm, Y = 169.0 mm, Z = 85.8 mm,
      W = 0.0 deg, P = 0.0 deg, R = 0.0 deg
   GP2:
       UF : 1, UT : 2,
      J1 = 0.0 deg, J2 = 0.0 deg
};
P[69] {
   GP1:
       UF : 5, UT : 6,     CONFIG: 'N U T, 0, 0, 0',
      X = 124.0 mm, Y = 173.0 mm, Z = 85.8 mm,
      W = 0.0 deg, P = 0.0 deg, R = 0.0 deg
   GP2:
       UF : 1, UT : 2,
      J1 = 0.0 deg, J2 = 0.0 deg
};
P[70] {
   GP1:
       UF : 5, UT : 6,     CONFIG: 'N U T, 0, 0, 0',
      X = 149.0 mm, Y = 148.0 mm, Z = 85.8 mm,
      W = 0.0 deg, P = 0.0 deg, R = 0.0 deg
   GP2:
       UF : 1, UT : 2,
      J1 = 0.0 deg, J2 = 0.0 deg
};
P[71] {
   GP1:
       UF : 5, UT : 6,     CONFIG: 'N U T, 0, 0, 0',
      X = 149.0 mm, Y = 153.0 mm, Z = 85.8 mm,
      W = 0.0 deg, P = 0.0 deg, R = 0.0 deg
   GP2:
       UF : 1, UT : 2,
      J1 = 0.0 deg, J2 = 0.0 deg
};
P[72] {
   GP1:
       UF : 5, UT : 6,     CONFIG: 'N U T, 0, 0, 0',
      X = 124.0 mm, Y = 178.0 mm, Z = 85.8 mm,
      W = 0.0 deg, P = 0.0 deg, R = 0.0 deg
   GP2:
       UF : 1, UT : 2,
      J1 = 0.0 deg, J2 = 0.0 deg
};
P[73] {
   GP1:
       UF : 5, UT : 6,     CONFIG: 'N U T, 0, 0, 0',
      X = 124.0 mm, Y = 183.0 mm, Z = 85.8 mm,
      W = 0.0 deg, P = 0.0 deg, R = 0.0 deg
   GP2:
       UF : 1, UT : 2,
      J1 = 0.0 deg, J2 = 0.0 deg
};
P[74] {
   GP1:
       UF : 5, UT : 6,     CONFIG: 'N U T, 0, 0, 0',
      X = 149.0 mm, Y = 158.0 mm, Z = 85.8 mm,
      W = 0.0 deg, P = 0.0 deg, R = 0.0 deg
   GP2:
       UF : 1, UT : 2,
      J1 = 0.0 deg, J2 = 0.0 deg
};
P[75] {
   GP1:
       UF : 5, UT : 6,     CONFIG: 'N U T, 0, 0, 0',
      X = 149.0 mm, Y = 162.0 mm, Z = 85.8 mm,
      W = 0.0 deg, P = 0.0 deg, R = 0.0 deg
   GP2:
       UF : 1, UT : 2,
      J1 = 0.0 deg, J2 = 0.0 deg
};
P[76] {
   GP1:
       UF : 5, UT : 6,     CONFIG: 'N U T, 0, 0, 0',
      X = 124.0 mm, Y = 188.0 mm, Z = 85.8 mm,
      W = 0.0 deg, P = 0.0 deg, R = 0.0 deg
   GP2:
       UF : 1, UT : 2,
      J1 = 0.0 deg, J2 = 0.0 deg
};
P[77] {
   GP1:
       UF : 5, UT : 6,     CONFIG: 'N U T, 0, 0, 0',
      X = 124.0 mm, Y = 192.0 mm, Z = 85.8 mm,
      W = 0.0 deg, P = 0.0 deg, R = 0.0 deg
   GP2:
       UF : 1, UT : 2,
      J1 = 0.0 deg, J2 = 0.0 deg
};
P[78] {
   GP1:
       UF : 5, UT : 6,     CONFIG: 'N U T, 0, 0, 0',
      X = 149.0 mm, Y = 167.0 mm, Z = 85.8 mm,
      W = 0.0 deg, P = 0.0 deg, R = 0.0 deg
   GP2:
       UF : 1, UT : 2,
      J1 = 0.0 deg, J2 = 0.0 deg
};
P[79] {
   GP1:
       UF : 5, UT : 6,     CONFIG: 'N U T, 0, 0, 0',
      X = 149.0 mm, Y = 172.0 mm, Z = 85.8 mm,
      W = 0.0 deg, P = 0.0 deg, R = 0.0 deg
   GP2:
       UF : 1, UT : 2,
      J1 = 0.0 deg, J2 = 0.0 deg
};
P[80] {
   GP1:
       UF : 5, UT : 6,     CONFIG: 'N U T, 0, 0, 0',
      X = 126.0 mm, Y = 195.0 mm, Z = 85.8 mm,
      W = 0.0 deg, P = 0.0 deg, R = 0.0 deg
   GP2:
       UF : 1, UT : 2,
      J1 = 0.0 deg, J2 = 0.0 deg
};
P[81] {
   GP1:
       UF : 5, UT : 6,     CONFIG: 'N U T, 0, 0, 0',
      X = 130.0 mm, Y = 195.0 mm, Z = 85.8 mm,
      W = 0.0 deg, P = 0.0 deg, R = 0.0 deg
   GP2:
       UF : 1, UT : 2,
      J1 = 0.0 deg, J2 = 0.0 deg
};
P[82] {
   GP1:
       UF : 5, UT : 6,     CONFIG: 'N U T, 0, 0, 0',
      X = 149.0 mm, Y = 176.0 mm, Z = 85.8 mm,
      W = 0.0 deg, P = 0.0 deg, R = 0.0 deg
   GP2:
       UF : 1, UT : 2,
      J1 = 0.0 deg, J2 = 0.0 deg
};
P[83] {
   GP1:
       UF : 5, UT : 6,     CONFIG: 'N U T, 0, 0, 0',
      X = 149.0 mm, Y = 181.0 mm, Z = 85.8 mm,
      W = 0.0 deg, P = 0.0 deg, R = 0.0 deg
   GP2:
       UF : 1, UT : 2,
      J1 = 0.0 deg, J2 = 0.0 deg
};
P[84] {
   GP1:
       UF : 5, UT : 6,     CONFIG: 'N U T, 0, 0, 0',
      X = 135.0 mm, Y = 195.0 mm, Z = 85.8 mm,
      W = 0.0 deg, P = 0.0 deg, R = 0.0 deg
   GP2:
       UF : 1, UT : 2,
      J1 = 0.0 deg, J2 = 0.0 deg
};
P[85] {
   GP1:
       UF : 5, UT : 6,     CONFIG: 'N U T, 0, 0, 0',
      X = 140.0 mm, Y = 195.0 mm, Z = 85.8 mm,
      W = 0.0 deg, P = 0.0 deg, R = 0.0 deg
   GP2:
       UF : 1, UT : 2,
      J1 = 0.0 deg, J2 = 0.0 deg
};
P[86] {
   GP1:
       UF : 5, UT : 6,     CONFIG: 'N U T, 0, 0, 0',
      X = 149.0 mm, Y = 186.0 mm, Z = 85.8 mm,
      W = 0.0 deg, P = 0.0 deg, R = 0.0 deg
   GP2:
       UF : 1, UT : 2,
      J1 = 0.0 deg, J2 = 0.0 deg
};
P[87] {
   GP1:
       UF : 5, UT : 6,     CONFIG: 'N U T, 0, 0, 0',
      X = 149.0 mm, Y = 190.0 mm, Z = 85.8 mm,
      W = 0.0 deg, P = 0.0 deg, R = 0.0 deg
   GP2:
       UF : 1, UT : 2,
      J1 = 0.0 deg, J2 = 0.0 deg
};
P[88] {
   GP1:
       UF : 5, UT : 6,     CONFIG: 'N U T, 0, 0, 0',
      X = 144.0 mm, Y = 195.0 mm, Z = 85.8 mm,
      W = 0.0 deg, P = 0.0 deg, R = 0.0 deg
   GP2:
       UF : 1, UT : 2,
      J1 = 0.0 deg, J2 = 0.0 deg
};
P[89] {
   GP1:
       UF : 5, UT : 6,     CONFIG: 'N U T, 0, 0, 0',
      X = -82.7 mm, Y = -29.3 mm, Z = 85.8 mm,
      W = 0.0 deg, P = 0.0 deg, R = 0.0 deg
   GP2:
       UF : 1, UT : 2,
      J1 = 0.0 deg, J2 = 0.0 deg
};
P[90] {
   GP1:
       UF : 5, UT : 6,     CONFIG: 'N U T, 0, 0, 0',
      X = -81.6 mm, Y = -30.4 mm, Z = 85.8 mm,
      W = 0.0 deg, P = 0.0 deg, R = 0.0 deg
   GP2:
       UF : 1, UT : 2,
      J1 = 0.0 deg, J2 = 0.0 deg
};
P[91] {
   GP1:
       UF : 5, UT : 6,     CONFIG: 'N U T, 0, 0, 0',
      X = -81.6 mm, Y = -35.1 mm, Z = 85.8 mm,
      W = 0.0 deg, P = 0.0 deg, R = 0.0 deg
   GP2:
       UF : 1, UT : 2,
      J1 = 0.0 deg, J2 = 0.0 deg
};
P[92] {
   GP1:
       UF : 5, UT : 6,     CONFIG: 'N U T, 0, 0, 0',
      X = -87.4 mm, Y = -29.3 mm, Z = 85.8 mm,
      W = 0.0 deg, P = 0.0 deg, R = 0.0 deg
   GP2:
       UF : 1, UT : 2,
      J1 = 0.0 deg, J2 = 0.0 deg
};
P[93] {
   GP1:
       UF : 5, UT : 6,     CONFIG: 'N U T, 0, 0, 0',
      X = -92.1 mm, Y = -29.3 mm, Z = 85.8 mm,
      W = 0.0 deg, P = 0.0 deg, R = 0.0 deg
   GP2:
       UF : 1, UT : 2,
      J1 = 0.0 deg, J2 = 0.0 deg
};
P[94] {
   GP1:
       UF : 5, UT : 6,     CONFIG: 'N U T, 0, 0, 0',
      X = 19.0 mm, Y = -140.0 mm, Z = 85.8 mm,
      W = 0.0 deg, P = 0.0 deg, R = 0.0 deg
   GP2:
       UF : 1, UT : 2,
      J1 = 0.0 deg, J2 = 0.0 deg
};
P[95] {
   GP1:
       UF : 5, UT : 6,     CONFIG: 'N U T, 0, 0, 0',
      X = 14.3 mm, Y = -140.0 mm, Z = 85.8 mm,
      W = 0.0 deg, P = 0.0 deg, R = 0.0 deg
   GP2:
       UF : 1, UT : 2,
      J1 = 0.0 deg, J2 = 0.0 deg
};
P[96] {
   GP1:
       UF : 5, UT : 6,     CONFIG: 'N U T, 0, 0, 0',
      X = -96.8 mm, Y = -29.3 mm, Z = 85.8 mm,
      W = 0.0 deg, P = 0.0 deg, R = 0.0 deg
   GP2:
       UF : 1, UT : 2,
      J1 = 0.0 deg, J2 = 0.0 deg
};
P[97] {
   GP1:
       UF : 5, UT : 6,     CONFIG: 'N U T, 0, 0, 0',
      X = -101.0 mm, Y = -29.3 mm, Z = 85.8 mm,
      W = 0.0 deg, P = 0.0 deg, R = 0.0 deg
   GP2:
       UF : 1, UT : 2,
      J1 = 0.0 deg, J2 = 0.0 deg
};
P[98] {
   GP1:
       UF : 5, UT : 6,     CONFIG: 'N U T, 0, 0, 0',
      X = 9.57 mm, Y = -140.0 mm, Z = 85.8 mm,
      W = 0.0 deg, P = 0.0 deg, R = 0.0 deg
   GP2:
       UF : 1, UT : 2,
      J1 = 0.0 deg, J2 = 0.0 deg
};
P[99] {
   GP1:
       UF : 5, UT : 6,     CONFIG: 'N U T, 0, 0, 0',
      X = 4.87 mm, Y = -140.0 mm, Z = 85.8 mm,
      W = 0.0 deg, P = 0.0 deg, R = 0.0 deg
   GP2:
       UF : 1, UT : 2,
      J1 = 0.0 deg, J2 = 0.0 deg
};
P[100] {
   GP1:
       UF : 5, UT : 6,     CONFIG: 'N U T, 0, 0, 0',
      X = -106.0 mm, Y = -29.3 mm, Z = 85.8 mm,
      W = 0.0 deg, P = 0.0 deg, R = 0.0 deg
   GP2:
       UF : 1, UT : 2,
      J1 = 0.0 deg, J2 = 0.0 deg
};
P[101] {
   GP1:
       UF : 5, UT : 6,     CONFIG: 'N U T, 0, 0, 0',
      X = -111.0 mm, Y = -29.3 mm, Z = 85.8 mm,
      W = 0.0 deg, P = 0.0 deg, R = 0.0 deg
   GP2:
       UF : 1, UT : 2,
      J1 = 0.0 deg, J2 = 0.0 deg
};
P[102] {
   GP1:
       UF : 5, UT : 6,     CONFIG: 'N U T, 0, 0, 0',
      X = 0.169 mm, Y = -140.0 mm, Z = 85.8 mm,
      W = 0.0 deg, P = 0.0 deg, R = 0.0 deg
   GP2:
       UF : 1, UT : 2,
      J1 = 0.0 deg, J2 = 0.0 deg
};
P[103] {
   GP1:
       UF : 5, UT : 6,     CONFIG: 'N U T, 0, 0, 0',
      X = -4.53 mm, Y = -140.0 mm, Z = 85.8 mm,
      W = 0.0 deg, P = 0.0 deg, R = 0.0 deg
   GP2:
       UF : 1, UT : 2,
      J1 = 0.0 deg, J2 = 0.0 deg
};
P[104] {
   GP1:
       UF : 5, UT : 6,     CONFIG: 'N U T, 0, 0, 0',
      X = -116.0 mm, Y = -29.3 mm, Z = 85.8 mm,
      W = 0.0 deg, P = 0.0 deg, R = 0.0 deg
   GP2:
       UF : 1, UT : 2,
      J1 = 0.0 deg, J2 = 0.0 deg
};
P[105] {
   GP1:
       UF : 5, UT : 6,     CONFIG: 'N U T, 0, 0, 0',
      X = -120.0 mm, Y = -29.3 mm, Z = 85.8 mm,
      W = 0.0 deg, P = 0.0 deg, R = 0.0 deg
   GP2:
       UF : 1, UT : 2,
      J1 = 0.0 deg, J2 = 0.0 deg
};
P[106] {
   GP1:
       UF : 5, UT : 6,     CONFIG: 'N U T, 0, 0, 0',
      X = -9.23 mm, Y = -140.0 mm, Z = 85.8 mm,
      W = 0.0 deg, P = 0.0 deg, R = 0.0 deg
   GP2:
       UF : 1, UT : 2,
      J1 = 0.0 deg, J2 = 0.0 deg
};
P[107] {
   GP1:
       UF : 5, UT : 6,     CONFIG: 'N U T, 0, 0, 0',
      X = -13.9 mm, Y = -140.0 mm, Z = 85.8 mm,
      W = 0.0 deg, P = 0.0 deg, R = 0.0 deg
   GP2:
       UF : 1, UT : 2,
      J1 = 0.0 deg, J2 = 0.0 deg
};
P[108] {
   GP1:
       UF : 5, UT : 6,     CONFIG: 'N U T, 0, 0, 0',
      X = -125.0 mm, Y = -29.3 mm, Z = 85.8 mm,
      W = 0.0 deg, P = 0.0 deg, R = 0.0 deg
   GP2:
       UF : 1, UT : 2,
      J1 = 0.0 deg, J2 = 0.0 deg
};
P[109] {
   GP1:
       UF : 5, UT : 6,     CONFIG: 'N U T, 0, 0, 0',
      X = -130.0 mm, Y = -29.3 mm, Z = 85.8 mm,
      W = 0.0 deg, P = 0.0 deg, R = 0.0 deg
   GP2:
       UF : 1, UT : 2,
      J1 = 0.0 deg, J2 = 0.0 deg
};
P[110] {
   GP1:
       UF : 5, UT : 6,     CONFIG: 'N U T, 0, 0, 0',
      X = -18.6 mm, Y = -140.0 mm, Z = 85.8 mm,
      W = 0.0 deg, P = 0.0 deg, R = 0.0 deg
   GP2:
       UF : 1, UT : 2,
      J1 = 0.0 deg, J2 = 0.0 deg
};
P[111] {
   GP1:
       UF : 5, UT : 6,     CONFIG: 'N U T, 0, 0, 0',
      X = -23.3 mm, Y = -140.0 mm, Z = 85.8 mm,
      W = 0.0 deg, P = 0.0 deg, R = 0.0 deg
   GP2:
       UF : 1, UT : 2,
      J1 = 0.0 deg, J2 = 0.0 deg
};
P[112] {
   GP1:
       UF : 5, UT : 6,     CONFIG: 'N U T, 0, 0, 0',
      X = -134.0 mm, Y = -29.3 mm, Z = 85.8 mm,
      W = 0.0 deg, P = 0.0 deg, R = 0.0 deg
   GP2:
       UF : 1, UT : 2,
      J1 = 0.0 deg, J2 = 0.0 deg
};
P[113] {
   GP1:
       UF : 5, UT : 6,     CONFIG: 'N U T, 0, 0, 0',
      X = -163.0 mm, Y = -75.6 mm, Z = 85.8 mm,
      W = 0.0 deg, P = 0.0 deg, R = 0.0 deg
   GP2:
       UF : 1, UT : 2,
      J1 = 0.0 deg, J2 = 0.0 deg
};
P[114] {
   GP1:
       UF : 5, UT : 6,     CONFIG: 'N U T, 0, 0, 0',
      X = -166.0 mm, Y = -72.6 mm, Z = 85.8 mm,
      W = 0.0 deg, P = 0.0 deg, R = 0.0 deg
   GP2:
       UF : 1, UT : 2,
      J1 = 0.0 deg, J2 = 0.0 deg
};
P[115] {
   GP1:
       UF : 5, UT : 6,     CONFIG: 'N U T, 0, 0, 0',
      X = -166.0 mm, Y = -67.9 mm, Z = 85.8 mm,
      W = 0.0 deg, P = 0.0 deg, R = 0.0 deg
   GP2:
       UF : 1, UT : 2,
      J1 = 0.0 deg, J2 = 0.0 deg
};
P[116] {
   GP1:
       UF : 5, UT : 6,     CONFIG: 'N U T, 0, 0, 0',
      X = -159.0 mm, Y = -74.9 mm, Z = 85.8 mm,
      W = 0.0 deg, P = 0.0 deg, R = 0.0 deg
   GP2:
       UF : 1, UT : 2,
      J1 = 0.0 deg, J2 = 0.0 deg
};
P[117] {
   GP1:
       UF : 5, UT : 6,     CONFIG: 'N U T, 0, 0, 0',
      X = -156.0 mm, Y = -73.9 mm, Z = 85.8 mm,
      W = 0.0 deg, P = 0.0 deg, R = 0.0 deg
   GP2:
       UF : 1, UT : 2,
      J1 = 0.0 deg, J2 = 0.0 deg
};
P[118] {
   GP1:
       UF : 5, UT : 6,     CONFIG: 'N U T, 0, 0, 0',
      X = -166.0 mm, Y = -63.2 mm, Z = 85.8 mm,
      W = 0.0 deg, P = 0.0 deg, R = 0.0 deg
   GP2:
       UF : 1, UT : 2,
      J1 = 0.0 deg, J2 = 0.0 deg
};
P[119] {
   GP1:
       UF : 5, UT : 6,     CONFIG: 'N U T, 0, 0, 0',
      X = -166.0 mm, Y = -58.5 mm, Z = 85.8 mm,
      W = 0.0 deg, P = 0.0 deg, R = 0.0 deg
   GP2:
       UF : 1, UT : 2,
      J1 = 0.0 deg, J2 = 0.0 deg
};
P[120] {
   GP1:
       UF : 5, UT : 6,     CONFIG: 'N U T, 0, 0, 0',
      X = -152.0 mm, Y = -72.9 mm, Z = 85.8 mm,
      W = 0.0 deg, P = 0.0 deg, R = 0.0 deg
   GP2:
       UF : 1, UT : 2,
      J1 = 0.0 deg, J2 = 0.0 deg
};
P[121] {
   GP1:
       UF : 5, UT : 6,     CONFIG: 'N U T, 0, 0, 0',
      X = -148.0 mm, Y = -71.9 mm, Z = 85.8 mm,
      W = 0.0 deg, P = 0.0 deg, R = 0.0 deg
   GP2:
       UF : 1, UT : 2,
      J1 = 0.0 deg, J2 = 0.0 deg
};
P[122] {
   GP1:
       UF : 5, UT : 6,     CONFIG: 'N U T, 0, 0, 0',
      X = -166.0 mm, Y = -53.8 mm, Z = 85.8 mm,
      W = 0.0 deg, P = 0.0 deg, R = 0.0 deg
   GP2:
       UF : 1, UT : 2,
      J1 = 0.0 deg, J2 = 0.0 deg
};
P[123] {
   GP1:
       UF : 5, UT : 6,     CONFIG: 'N U T, 0, 0, 0',
      X = -166.0 mm, Y = -49.1 mm, Z = 85.8 mm,
      W = 0.0 deg, P = 0.0 deg, R = 0.0 deg
   GP2:
       UF : 1, UT : 2,
      J1 = 0.0 deg, J2 = 0.0 deg
};
P[124] {
   GP1:
       UF : 5, UT : 6,     CONFIG: 'N U T, 0, 0, 0',
      X = -144.0 mm, Y = -70.9 mm, Z = 85.8 mm,
      W = 0.0 deg, P = 0.0 deg, R = 0.0 deg
   GP2:
       UF : 1, UT : 2,
      J1 = 0.0 deg, J2 = 0.0 deg
};
P[125] {
   GP1:
       UF : 5, UT : 6,     CONFIG: 'N U T, 0, 0, 0',
      X = -141.0 mm, Y = -69.9 mm, Z = 85.8 mm,
      W = 0.0 deg, P = 0.0 deg, R = 0.0 deg
   GP2:
       UF : 1, UT : 2,
      J1 = 0.0 deg, J2 = 0.0 deg
};
P[126] {
   GP1:
       UF : 5, UT : 6,     CONFIG: 'N U T, 0, 0, 0',
      X = -166.0 mm, Y = -44.4 mm, Z = 85.8 mm,
      W = 0.0 deg, P = 0.0 deg, R = 0.0 deg
   GP2:
       UF : 1, UT : 2,
      J1 = 0.0 deg, J2 = 0.0 deg
};
P[127] {
   GP1:
       UF : 5, UT : 6,     CONFIG: 'N U T, 0, 0, 0',
      X = -166.0 mm, Y = -39.7 mm, Z = 85.8 mm,
      W = 0.0 deg, P = 0.0 deg, R = 0.0 deg
   GP2:
       UF : 1, UT : 2,
      J1 = 0.0 deg, J2 = 0.0 deg
};
P[128] {
   GP1:
       UF : 5, UT : 6,     CONFIG: 'N U T, 0, 0, 0',
      X = -137.0 mm, Y = -68.9 mm, Z = 85.8 mm,
      W = 0.0 deg, P = 0.0 deg, R = 0.0 deg
   GP2:
       UF : 1, UT : 2,
      J1 = 0.0 deg, J2 = 0.0 deg
};
P[129] {
   GP1:
       UF : 5, UT : 6,     CONFIG: 'N U T, 0, 0, 0',
      X = -133.0 mm, Y = -67.9 mm, Z = 85.8 mm,
      W = 0.0 deg, P = 0.0 deg, R = 0.0 deg
   GP2:
       UF : 1, UT : 2,
      J1 = 0.0 deg, J2 = 0.0 deg
};
P[130] {
   GP1:
       UF : 5, UT : 6,     CONFIG: 'N U T, 0, 0, 0',
      X = -166.0 mm, Y = -35.0 mm, Z = 85.8 mm,
      W = 0.0 deg, P = 0.0 deg, R = 0.0 deg
   GP2:
       UF : 1, UT : 2,
      J1 = 0.0 deg, J2 = 0.0 deg
};
P[131] {
   GP1:
       UF : 5, UT : 6,     CONFIG: 'N U T, 0, 0, 0',
      X = -166.0 mm, Y = -30.3 mm, Z = 85.8 mm,
      W = 0.0 deg, P = 0.0 deg, R = 0.0 deg
   GP2:
       UF : 1, UT : 2,
      J1 = 0.0 deg, J2 = 0.0 deg
};
P[132] {
   GP1:
       UF : 5, UT : 6,     CONFIG: 'N U T, 0, 0, 0',
      X = -130.0 mm, Y = -66.9 mm, Z = 85.8 mm,
      W = 0.0 deg, P = 0.0 deg, R = 0.0 deg
   GP2:
       UF : 1, UT : 2,
      J1 = 0.0 deg, J2 = 0.0 deg
};
P[133] {
   GP1:
       UF : 5, UT : 6,     CONFIG: 'N U T, 0, 0, 0',
      X = -126.0 mm, Y = -65.9 mm, Z = 85.8 mm,
      W = 0.0 deg, P = 0.0 deg, R = 0.0 deg
   GP2:
       UF : 1, UT : 2,
      J1 = 0.0 deg, J2 = 0.0 deg
};
P[134] {
   GP1:
       UF : 5, UT : 6,     CONFIG: 'N U T, 0, 0, 0',
      X = -163.0 mm, Y = -29.3 mm, Z = 85.8 mm,
      W = 0.0 deg, P = 0.0 deg, R = 0.0 deg
   GP2:
       UF : 1, UT : 2,
      J1 = 0.0 deg, J2 = 0.0 deg
};
P[135] {
   GP1:
       UF : 5, UT : 6,     CONFIG: 'N U T, 0, 0, 0',
      X = -160.0 mm, Y = -29.3 mm, Z = 85.8 mm,
      W = 0.0 deg, P = 0.0 deg, R = 0.0 deg
   GP2:
       UF : 1, UT : 2,
      J1 = 0.0 deg, J2 = 0.0 deg
};
P[136] {
   GP1:
       UF : 5, UT : 6,     CONFIG: 'N U T, 0, 0, 0',
      X = -160.0 mm, Y = -29.3 mm, Z = 85.8 mm,
      W = 0.0 deg, P = 0.0 deg, R = 0.0 deg
   GP2:
       UF : 1, UT : 2,
      J1 = 0.0 deg, J2 = 0.0 deg
};
P[137] {
   GP1:
       UF : 5, UT : 6,     CONFIG: 'N U T, 0, 0, 0',
      X = -158.0 mm, Y = -29.3 mm, Z = 85.8 mm,
      W = 0.0 deg, P = 0.0 deg, R = 0.0 deg
   GP2:
       UF : 1, UT : 2,
      J1 = 0.0 deg, J2 = 0.0 deg
};
P[138] {
   GP1:
       UF : 5, UT : 6,     CONFIG: 'N U T, 0, 0, 0',
      X = -122.0 mm, Y = -64.9 mm, Z = 85.8 mm,
      W = 0.0 deg, P = 0.0 deg, R = 0.0 deg
   GP2:
       UF : 1, UT : 2,
      J1 = 0.0 deg, J2 = 0.0 deg
};
P[139] {
   GP1:
       UF : 5, UT : 6,     CONFIG: 'N U T, 0, 0, 0',
      X = -119.0 mm, Y = -63.9 mm, Z = 85.8 mm,
      W = 0.0 deg, P = 0.0 deg, R = 0.0 deg
   GP2:
       UF : 1, UT : 2,
      J1 = 0.0 deg, J2 = 0.0 deg
};
P[140] {
   GP1:
       UF : 5, UT : 6,     CONFIG: 'N U T, 0, 0, 0',
      X = -153.0 mm, Y = -29.3 mm, Z = 85.8 mm,
      W = 0.0 deg, P = 0.0 deg, R = 0.0 deg
   GP2:
       UF : 1, UT : 2,
      J1 = 0.0 deg, J2 = 0.0 deg
};
P[141] {
   GP1:
       UF : 5, UT : 6,     CONFIG: 'N U T, 0, 0, 0',
      X = -149.0 mm, Y = -29.3 mm, Z = 85.8 mm,
      W = 0.0 deg, P = 0.0 deg, R = 0.0 deg
   GP2:
       UF : 1, UT : 2,
      J1 = 0.0 deg, J2 = 0.0 deg
};
P[142] {
   GP1:
       UF : 5, UT : 6,     CONFIG: 'N U T, 0, 0, 0',
      X = -115.0 mm, Y = -62.9 mm, Z = 85.8 mm,
      W = 0.0 deg, P = 0.0 deg, R = 0.0 deg
   GP2:
       UF : 1, UT : 2,
      J1 = 0.0 deg, J2 = 0.0 deg
};
P[143] {
   GP1:
       UF : 5, UT : 6,     CONFIG: 'N U T, 0, 0, 0',
      X = -113.0 mm, Y = -62.5 mm, Z = 85.8 mm,
      W = 0.0 deg, P = 0.0 deg, R = 0.0 deg
   GP2:
       UF : 1, UT : 2,
      J1 = 0.0 deg, J2 = 0.0 deg
};
P[144] {
   GP1:
       UF : 5, UT : 6,     CONFIG: 'N U T, 0, 0, 0',
      X = -112.0 mm, Y = -62.2 mm, Z = 85.8 mm,
      W = 0.0 deg, P = 0.0 deg, R = 0.0 deg
   GP2:
       UF : 1, UT : 2,
      J1 = 0.0 deg, J2 = 0.0 deg
};
P[145] {
   GP1:
       UF : 5, UT : 6,     CONFIG: 'N U T, 0, 0, 0',
      X = -111.0 mm, Y = -62.1 mm, Z = 85.8 mm,
      W = 0.0 deg, P = 0.0 deg, R = 0.0 deg
   GP2:
       UF : 1, UT : 2,
      J1 = 0.0 deg, J2 = 0.0 deg
};
P[146] {
   GP1:
       UF : 5, UT : 6,     CONFIG: 'N U T, 0, 0, 0',
      X = -144.0 mm, Y = -29.3 mm, Z = 85.8 mm,
      W = 0.0 deg, P = 0.0 deg, R = 0.0 deg
   GP2:
       UF : 1, UT : 2,
      J1 = 0.0 deg, J2 = 0.0 deg
};
P[147] {
   GP1:
       UF : 5, UT : 6,     CONFIG: 'N U T, 0, 0, 0',
      X = -139.0 mm, Y = -29.3 mm, Z = 85.8 mm,
      W = 0.0 deg, P = 0.0 deg, R = 0.0 deg
   GP2:
       UF : 1, UT : 2,
      J1 = 0.0 deg, J2 = 0.0 deg
};
P[148] {
   GP1:
       UF : 5, UT : 6,     CONFIG: 'N U T, 0, 0, 0',
      X = -105.0 mm, Y = -63.8 mm, Z = 85.8 mm,
      W = 0.0 deg, P = 0.0 deg, R = 0.0 deg
   GP2:
       UF : 1, UT : 2,
      J1 = 0.0 deg, J2 = 0.0 deg
};
P[149] {
   GP1:
       UF : 5, UT : 6,     CONFIG: 'N U T, 0, 0, 0',
      X = -104.0 mm, Y = -64.0 mm, Z = 85.8 mm,
      W = 0.0 deg, P = 0.0 deg, R = 0.0 deg
   GP2:
       UF : 1, UT : 2,
      J1 = 0.0 deg, J2 = 0.0 deg
};
P[150] {
   GP1:
       UF : 5, UT : 6,     CONFIG: 'N U T, 0, 0, 0',
      X = -103.0 mm, Y = -64.8 mm, Z = 85.8 mm,
      W = 0.0 deg, P = 0.0 deg, R = 0.0 deg
   GP2:
       UF : 1, UT : 2,
      J1 = 0.0 deg, J2 = 0.0 deg
};
P[151] {
   GP1:
       UF : 5, UT : 6,     CONFIG: 'N U T, 0, 0, 0',
      X = -102.0 mm, Y = -65.8 mm, Z = 85.8 mm,
      W = 0.0 deg, P = 0.0 deg, R = 0.0 deg
   GP2:
       UF : 1, UT : 2,
      J1 = 0.0 deg, J2 = 0.0 deg
};
P[152] {
   GP1:
       UF : 5, UT : 6,     CONFIG: 'N U T, 0, 0, 0',
      X = -101.0 mm, Y = -66.9 mm, Z = 85.8 mm,
      W = 0.0 deg, P = 0.0 deg, R = 0.0 deg
   GP2:
       UF : 1, UT : 2,
      J1 = 0.0 deg, J2 = 0.0 deg
};
P[153] {
   GP1:
       UF : 5, UT : 6,     CONFIG: 'N U T, 0, 0, 0',
      X = -101.0 mm, Y = -67.3 mm, Z = 85.8 mm,
      W = 0.0 deg, P = 0.0 deg, R = 0.0 deg
   GP2:
       UF : 1, UT : 2,
      J1 = 0.0 deg, J2 = 0.0 deg
};
P[154] {
   GP1:
       UF : 5, UT : 6,     CONFIG: 'N U T, 0, 0, 0',
      X = -28.0 mm, Y = -140.0 mm, Z = 85.8 mm,
      W = 0.0 deg, P = 0.0 deg, R = 0.0 deg
   GP2:
       UF : 1, UT : 2,
      J1 = 0.0 deg, J2 = 0.0 deg
};
P[155] {
   GP1:
       UF : 5, UT : 6,     CONFIG: 'N U T, 0, 0, 0',
      X = -32.7 mm, Y = -140.0 mm, Z = 85.8 mm,
      W = 0.0 deg, P = 0.0 deg, R = 0.0 deg
   GP2:
       UF : 1, UT : 2,
      J1 = 0.0 deg, J2 = 0.0 deg
};
P[156] {
   GP1:
       UF : 5, UT : 6,     CONFIG: 'N U T, 0, 0, 0',
      X = -98.6 mm, Y = -74.5 mm, Z = 85.8 mm,
      W = 0.0 deg, P = 0.0 deg, R = 0.0 deg
   GP2:
       UF : 1, UT : 2,
      J1 = 0.0 deg, J2 = 0.0 deg
};
P[157] {
   GP1:
       UF : 5, UT : 6,     CONFIG: 'N U T, 0, 0, 0',
      X = -96.9 mm, Y = -80.9 mm, Z = 85.8 mm,
      W = 0.0 deg, P = 0.0 deg, R = 0.0 deg
   GP2:
       UF : 1, UT : 2,
      J1 = 0.0 deg, J2 = 0.0 deg
};
P[158] {
   GP1:
       UF : 5, UT : 6,     CONFIG: 'N U T, 0, 0, 0',
      X = -37.4 mm, Y = -140.0 mm, Z = 85.8 mm,
      W = 0.0 deg, P = 0.0 deg, R = 0.0 deg
   GP2:
       UF : 1, UT : 2,
      J1 = 0.0 deg, J2 = 0.0 deg
};
P[159] {
   GP1:
       UF : 5, UT : 6,     CONFIG: 'N U T, 0, 0, 0',
      X = -42.2 mm, Y = -140.0 mm, Z = 85.8 mm,
      W = 0.0 deg, P = 0.0 deg, R = 0.0 deg
   GP2:
       UF : 1, UT : 2,
      J1 = 0.0 deg, J2 = 0.0 deg
};
P[160] {
   GP1:
       UF : 5, UT : 6,     CONFIG: 'N U T, 0, 0, 0',
      X = -95.4 mm, Y = -87.1 mm, Z = 85.8 mm,
      W = 0.0 deg, P = 0.0 deg, R = 0.0 deg
   GP2:
       UF : 1, UT : 2,
      J1 = 0.0 deg, J2 = 0.0 deg
};
P[161] {
   GP1:
       UF : 5, UT : 6,     CONFIG: 'N U T, 0, 0, 0',
      X = -95.3 mm, Y = -88.1 mm, Z = 85.8 mm,
      W = 0.0 deg, P = 0.0 deg, R = 0.0 deg
   GP2:
       UF : 1, UT : 2,
      J1 = 0.0 deg, J2 = 0.0 deg
};
P[162] {
   GP1:
       UF : 5, UT : 6,     CONFIG: 'N U T, 0, 0, 0',
      X = -95.4 mm, Y = -89.5 mm, Z = 85.8 mm,
      W = 0.0 deg, P = 0.0 deg, R = 0.0 deg
   GP2:
       UF : 1, UT : 2,
      J1 = 0.0 deg, J2 = 0.0 deg
};
P[163] {
   GP1:
       UF : 5, UT : 6,     CONFIG: 'N U T, 0, 0, 0',
      X = -95.6 mm, Y = -90.9 mm, Z = 85.8 mm,
      W = 0.0 deg, P = 0.0 deg, R = 0.0 deg
   GP2:
       UF : 1, UT : 2,
      J1 = 0.0 deg, J2 = 0.0 deg
};
P[164] {
   GP1:
       UF : 5, UT : 6,     CONFIG: 'N U T, 0, 0, 0',
      X = -95.8 mm, Y = -91.4 mm, Z = 85.8 mm,
      W = 0.0 deg, P = 0.0 deg, R = 0.0 deg
   GP2:
       UF : 1, UT : 2,
      J1 = 0.0 deg, J2 = 0.0 deg
};
P[165] {
   GP1:
       UF : 5, UT : 6,     CONFIG: 'N U T, 0, 0, 0',
      X = -46.9 mm, Y = -140.0 mm, Z = 85.8 mm,
      W = 0.0 deg, P = 0.0 deg, R = 0.0 deg
   GP2:
       UF : 1, UT : 2,
      J1 = 0.0 deg, J2 = 0.0 deg
};
P[166] {
   GP1:
       UF : 5, UT : 6,     CONFIG: 'N U T, 0, 0, 0',
      X = -51.6 mm, Y = -140.0 mm, Z = 85.8 mm,
      W = 0.0 deg, P = 0.0 deg, R = 0.0 deg
   GP2:
       UF : 1, UT : 2,
      J1 = 0.0 deg, J2 = 0.0 deg
};
P[167] {
   GP1:
       UF : 5, UT : 6,     CONFIG: 'N U T, 0, 0, 0',
      X = -97.2 mm, Y = -94.7 mm, Z = 85.8 mm,
      W = 0.0 deg, P = 0.0 deg, R = 0.0 deg
   GP2:
       UF : 1, UT : 2,
      J1 = 0.0 deg, J2 = 0.0 deg
};
P[168] {
   GP1:
       UF : 5, UT : 6,     CONFIG: 'N U T, 0, 0, 0',
      X = -97.3 mm, Y = -94.7 mm, Z = 85.8 mm,
      W = 0.0 deg, P = 0.0 deg, R = 0.0 deg
   GP2:
       UF : 1, UT : 2,
      J1 = 0.0 deg, J2 = 0.0 deg
};
P[169] {
   GP1:
       UF : 5, UT : 6,     CONFIG: 'N U T, 0, 0, 0',
      X = -98.5 mm, Y = -96.3 mm, Z = 85.8 mm,
      W = 0.0 deg, P = 0.0 deg, R = 0.0 deg
   GP2:
       UF : 1, UT : 2,
      J1 = 0.0 deg, J2 = 0.0 deg
};
P[170] {
   GP1:
       UF : 5, UT : 6,     CONFIG: 'N U T, 0, 0, 0',
      X = -100.0 mm, Y = -96.3 mm, Z = 85.8 mm,
      W = 0.0 deg, P = 0.0 deg, R = 0.0 deg
   GP2:
       UF : 1, UT : 2,
      J1 = 0.0 deg, J2 = 0.0 deg
};
P[171] {
   GP1:
       UF : 5, UT : 6,     CONFIG: 'N U T, 0, 0, 0',
      X = -56.3 mm, Y = -140.0 mm, Z = 85.8 mm,
      W = 0.0 deg, P = 0.0 deg, R = 0.0 deg
   GP2:
       UF : 1, UT : 2,
      J1 = 0.0 deg, J2 = 0.0 deg
};
P[172] {
   GP1:
       UF : 5, UT : 6,     CONFIG: 'N U T, 0, 0, 0',
      X = -61.0 mm, Y = -140.0 mm, Z = 85.8 mm,
      W = 0.0 deg, P = 0.0 deg, R = 0.0 deg
   GP2:
       UF : 1, UT : 2,
      J1 = 0.0 deg, J2 = 0.0 deg
};
P[173] {
   GP1:
       UF : 5, UT : 6,     CONFIG: 'N U T, 0, 0, 0',
      X = -105.0 mm, Y = -96.3 mm, Z = 85.8 mm,
      W = 0.0 deg, P = 0.0 deg, R = 0.0 deg
   GP2:
       UF : 1, UT : 2,
      J1 = 0.0 deg, J2 = 0.0 deg
};
P[174] {
   GP1:
       UF : 5, UT : 6,     CONFIG: 'N U T, 0, 0, 0',
      X = -110.0 mm, Y = -96.3 mm, Z = 85.8 mm,
      W = 0.0 deg, P = 0.0 deg, R = 0.0 deg
   GP2:
       UF : 1, UT : 2,
      J1 = 0.0 deg, J2 = 0.0 deg
};
P[175] {
   GP1:
       UF : 5, UT : 6,     CONFIG: 'N U T, 0, 0, 0',
      X = -65.7 mm, Y = -140.0 mm, Z = 85.8 mm,
      W = 0.0 deg, P = 0.0 deg, R = 0.0 deg
   GP2:
       UF : 1, UT : 2,
      J1 = 0.0 deg, J2 = 0.0 deg
};
P[176] {
   GP1:
       UF : 5, UT : 6,     CONFIG: 'N U T, 0, 0, 0',
      X = -70.4 mm, Y = -140.0 mm, Z = 85.8 mm,
      W = 0.0 deg, P = 0.0 deg, R = 0.0 deg
   GP2:
       UF : 1, UT : 2,
      J1 = 0.0 deg, J2 = 0.0 deg
};
P[177] {
   GP1:
       UF : 5, UT : 6,     CONFIG: 'N U T, 0, 0, 0',
      X = -114.0 mm, Y = -96.3 mm, Z = 85.8 mm,
      W = 0.0 deg, P = 0.0 deg, R = 0.0 deg
   GP2:
       UF : 1, UT : 2,
      J1 = 0.0 deg, J2 = 0.0 deg
};
P[178] {
   GP1:
       UF : 5, UT : 6,     CONFIG: 'N U T, 0, 0, 0',
      X = -119.0 mm, Y = -96.3 mm, Z = 85.8 mm,
      W = 0.0 deg, P = 0.0 deg, R = 0.0 deg
   GP2:
       UF : 1, UT : 2,
      J1 = 0.0 deg, J2 = 0.0 deg
};
P[179] {
   GP1:
       UF : 5, UT : 6,     CONFIG: 'N U T, 0, 0, 0',
      X = -75.1 mm, Y = -140.0 mm, Z = 85.8 mm,
      W = 0.0 deg, P = 0.0 deg, R = 0.0 deg
   GP2:
       UF : 1, UT : 2,
      J1 = 0.0 deg, J2 = 0.0 deg
};
P[180] {
   GP1:
       UF : 5, UT : 6,     CONFIG: 'N U T, 0, 0, 0',
      X = -79.8 mm, Y = -140.0 mm, Z = 85.8 mm,
      W = 0.0 deg, P = 0.0 deg, R = 0.0 deg
   GP2:
       UF : 1, UT : 2,
      J1 = 0.0 deg, J2 = 0.0 deg
};
P[181] {
   GP1:
       UF : 5, UT : 6,     CONFIG: 'N U T, 0, 0, 0',
      X = -124.0 mm, Y = -96.3 mm, Z = 85.8 mm,
      W = 0.0 deg, P = 0.0 deg, R = 0.0 deg
   GP2:
       UF : 1, UT : 2,
      J1 = 0.0 deg, J2 = 0.0 deg
};
P[182] {
   GP1:
       UF : 5, UT : 6,     CONFIG: 'N U T, 0, 0, 0',
      X = -129.0 mm, Y = -96.3 mm, Z = 85.8 mm,
      W = 0.0 deg, P = 0.0 deg, R = 0.0 deg
   GP2:
       UF : 1, UT : 2,
      J1 = 0.0 deg, J2 = 0.0 deg
};
P[183] {
   GP1:
       UF : 5, UT : 6,     CONFIG: 'N U T, 0, 0, 0',
      X = -84.5 mm, Y = -140.0 mm, Z = 85.8 mm,
      W = 0.0 deg, P = 0.0 deg, R = 0.0 deg
   GP2:
       UF : 1, UT : 2,
      J1 = 0.0 deg, J2 = 0.0 deg
};
P[184] {
   GP1:
       UF : 5, UT : 6,     CONFIG: 'N U T, 0, 0, 0',
      X = -89.2 mm, Y = -140.0 mm, Z = 85.8 mm,
      W = 0.0 deg, P = 0.0 deg, R = 0.0 deg
   GP2:
       UF : 1, UT : 2,
      J1 = 0.0 deg, J2 = 0.0 deg
};
P[185] {
   GP1:
       UF : 5, UT : 6,     CONFIG: 'N U T, 0, 0, 0',
      X = -133.0 mm, Y = -96.6 mm, Z = 85.8 mm,
      W = 0.0 deg, P = 0.0 deg, R = 0.0 deg
   GP2:
       UF : 1, UT : 2,
      J1 = 0.0 deg, J2 = 0.0 deg
};
P[186] {
   GP1:
       UF : 5, UT : 6,     CONFIG: 'N U T, 0, 0, 0',
      X = -133.0 mm, Y = -101.0 mm, Z = 85.8 mm,
      W = 0.0 deg, P = 0.0 deg, R = 0.0 deg
   GP2:
       UF : 1, UT : 2,
      J1 = 0.0 deg, J2 = 0.0 deg
};
P[187] {
   GP1:
       UF : 5, UT : 6,     CONFIG: 'N U T, 0, 0, 0',
      X = -93.9 mm, Y = -140.0 mm, Z = 85.8 mm,
      W = 0.0 deg, P = 0.0 deg, R = 0.0 deg
   GP2:
       UF : 1, UT : 2,
      J1 = 0.0 deg, J2 = 0.0 deg
};
P[188] {
   GP1:
       UF : 5, UT : 6,     CONFIG: 'N U T, 0, 0, 0',
      X = -98.6 mm, Y = -140.0 mm, Z = 85.8 mm,
      W = 0.0 deg, P = 0.0 deg, R = 0.0 deg
   GP2:
       UF : 1, UT : 2,
      J1 = 0.0 deg, J2 = 0.0 deg
};
P[189] {
   GP1:
       UF : 5, UT : 6,     CONFIG: 'N U T, 0, 0, 0',
      X = -133.0 mm, Y = -106.0 mm, Z = 85.8 mm,
      W = 0.0 deg, P = 0.0 deg, R = 0.0 deg
   GP2:
       UF : 1, UT : 2,
      J1 = 0.0 deg, J2 = 0.0 deg
};
P[190] {
   GP1:
       UF : 5, UT : 6,     CONFIG: 'N U T, 0, 0, 0',
      X = -133.0 mm, Y = -107.0 mm, Z = 85.8 mm,
      W = 0.0 deg, P = 0.0 deg, R = 0.0 deg
   GP2:
       UF : 1, UT : 2,
      J1 = 0.0 deg, J2 = 0.0 deg
};
P[191] {
   GP1:
       UF : 5, UT : 6,     CONFIG: 'N U T, 0, 0, 0',
      X = -136.0 mm, Y = -108.0 mm, Z = 85.8 mm,
      W = 0.0 deg, P = 0.0 deg, R = 0.0 deg
   GP2:
       UF : 1, UT : 2,
      J1 = 0.0 deg, J2 = 0.0 deg
};
P[192] {
   GP1:
       UF : 5, UT : 6,     CONFIG: 'N U T, 0, 0, 0',
      X = -103.0 mm, Y = -140.0 mm, Z = 85.8 mm,
      W = 0.0 deg, P = 0.0 deg, R = 0.0 deg
   GP2:
       UF : 1, UT : 2,
      J1 = 0.0 deg, J2 = 0.0 deg
};
P[193] {
   GP1:
       UF : 5, UT : 6,     CONFIG: 'N U T, 0, 0, 0',
      X = -108.0 mm, Y = -140.0 mm, Z = 85.8 mm,
      W = 0.0 deg, P = 0.0 deg, R = 0.0 deg
   GP2:
       UF : 1, UT : 2,
      J1 = 0.0 deg, J2 = 0.0 deg
};
P[194] {
   GP1:
       UF : 5, UT : 6,     CONFIG: 'N U T, 0, 0, 0',
      X = -139.0 mm, Y = -109.0 mm, Z = 85.8 mm,
      W = 0.0 deg, P = 0.0 deg, R = 0.0 deg
   GP2:
       UF : 1, UT : 2,
      J1 = 0.0 deg, J2 = 0.0 deg
};
P[195] {
   GP1:
       UF : 5, UT : 6,     CONFIG: 'N U T, 0, 0, 0',
      X = -143.0 mm, Y = -110.0 mm, Z = 85.8 mm,
      W = 0.0 deg, P = 0.0 deg, R = 0.0 deg
   GP2:
       UF : 1, UT : 2,
      J1 = 0.0 deg, J2 = 0.0 deg
};
P[196] {
   GP1:
       UF : 5, UT : 6,     CONFIG: 'N U T, 0, 0, 0',
      X = -113.0 mm, Y = -140.0 mm, Z = 85.8 mm,
      W = 0.0 deg, P = 0.0 deg, R = 0.0 deg
   GP2:
       UF : 1, UT : 2,
      J1 = 0.0 deg, J2 = 0.0 deg
};
P[197] {
   GP1:
       UF : 5, UT : 6,     CONFIG: 'N U T, 0, 0, 0',
      X = -117.0 mm, Y = -140.0 mm, Z = 85.8 mm,
      W = 0.0 deg, P = 0.0 deg, R = 0.0 deg
   GP2:
       UF : 1, UT : 2,
      J1 = 0.0 deg, J2 = 0.0 deg
};
P[198] {
   GP1:
       UF : 5, UT : 6,     CONFIG: 'N U T, 0, 0, 0',
      X = -147.0 mm, Y = -111.0 mm, Z = 85.8 mm,
      W = 0.0 deg, P = 0.0 deg, R = 0.0 deg
   GP2:
       UF : 1, UT : 2,
      J1 = 0.0 deg, J2 = 0.0 deg
};
P[199] {
   GP1:
       UF : 5, UT : 6,     CONFIG: 'N U T, 0, 0, 0',
      X = -150.0 mm, Y = -112.0 mm, Z = 85.8 mm,
      W = 0.0 deg, P = 0.0 deg, R = 0.0 deg
   GP2:
       UF : 1, UT : 2,
      J1 = 0.0 deg, J2 = 0.0 deg
};
P[200] {
   GP1:
       UF : 5, UT : 6,     CONFIG: 'N U T, 0, 0, 0',
      X = -122.0 mm, Y = -140.0 mm, Z = 85.8 mm,
      W = 0.0 deg, P = 0.0 deg, R = 0.0 deg
   GP2:
       UF : 1, UT : 2,
      J1 = 0.0 deg, J2 = 0.0 deg
};
P[201] {
   GP1:
       UF : 5, UT : 6,     CONFIG: 'N U T, 0, 0, 0',
      X = -127.0 mm, Y = -140.0 mm, Z = 85.8 mm,
      W = 0.0 deg, P = 0.0 deg, R = 0.0 deg
   GP2:
       UF : 1, UT : 2,
      J1 = 0.0 deg, J2 = 0.0 deg
};
P[202] {
   GP1:
       UF : 5, UT : 6,     CONFIG: 'N U T, 0, 0, 0',
      X = -154.0 mm, Y = -113.0 mm, Z = 85.8 mm,
      W = 0.0 deg, P = 0.0 deg, R = 0.0 deg
   GP2:
       UF : 1, UT : 2,
      J1 = 0.0 deg, J2 = 0.0 deg
};
P[203] {
   GP1:
       UF : 5, UT : 6,     CONFIG: 'N U T, 0, 0, 0',
      X = -157.0 mm, Y = -114.0 mm, Z = 85.8 mm,
      W = 0.0 deg, P = 0.0 deg, R = 0.0 deg
   GP2:
       UF : 1, UT : 2,
      J1 = 0.0 deg, J2 = 0.0 deg
};
P[204] {
   GP1:
       UF : 5, UT : 6,     CONFIG: 'N U T, 0, 0, 0',
      X = -157.0 mm, Y = -115.0 mm, Z = 85.8 mm,
      W = 0.0 deg, P = 0.0 deg, R = 0.0 deg
   GP2:
       UF : 1, UT : 2,
      J1 = 0.0 deg, J2 = 0.0 deg
};
P[205] {
   GP1:
       UF : 5, UT : 6,     CONFIG: 'N U T, 0, 0, 0',
      X = -131.0 mm, Y = -140.0 mm, Z = 85.8 mm,
      W = 0.0 deg, P = 0.0 deg, R = 0.0 deg
   GP2:
       UF : 1, UT : 2,
      J1 = 0.0 deg, J2 = 0.0 deg
};
P[206] {
   GP1:
       UF : 5, UT : 6,     CONFIG: 'N U T, 0, 0, 0',
      X = -136.0 mm, Y = -140.0 mm, Z = 85.8 mm,
      W = 0.0 deg, P = 0.0 deg, R = 0.0 deg
   GP2:
       UF : 1, UT : 2,
      J1 = 0.0 deg, J2 = 0.0 deg
};
P[207] {
   GP1:
       UF : 5, UT : 6,     CONFIG: 'N U T, 0, 0, 0',
      X = -157.0 mm, Y = -120.0 mm, Z = 85.8 mm,
      W = 0.0 deg, P = 0.0 deg, R = 0.0 deg
   GP2:
       UF : 1, UT : 2,
      J1 = 0.0 deg, J2 = 0.0 deg
};
P[208] {
   GP1:
       UF : 5, UT : 6,     CONFIG: 'N U T, 0, 0, 0',
      X = -157.0 mm, Y = -124.0 mm, Z = 85.8 mm,
      W = 0.0 deg, P = 0.0 deg, R = 0.0 deg
   GP2:
       UF : 1, UT : 2,
      J1 = 0.0 deg, J2 = 0.0 deg
};
P[209] {
   GP1:
       UF : 5, UT : 6,     CONFIG: 'N U T, 0, 0, 0',
      X = -141.0 mm, Y = -140.0 mm, Z = 85.8 mm,
      W = 0.0 deg, P = 0.0 deg, R = 0.0 deg
   GP2:
       UF : 1, UT : 2,
      J1 = 0.0 deg, J2 = 0.0 deg
};
P[210] {
   GP1:
       UF : 5, UT : 6,     CONFIG: 'N U T, 0, 0, 0',
      X = -146.0 mm, Y = -140.0 mm, Z = 85.8 mm,
      W = 0.0 deg, P = 0.0 deg, R = 0.0 deg
   GP2:
       UF : 1, UT : 2,
      J1 = 0.0 deg, J2 = 0.0 deg
};
P[211] {
   GP1:
       UF : 5, UT : 6,     CONFIG: 'N U T, 0, 0, 0',
      X = -157.0 mm, Y = -129.0 mm, Z = 85.8 mm,
      W = 0.0 deg, P = 0.0 deg, R = 0.0 deg
   GP2:
       UF : 1, UT : 2,
      J1 = 0.0 deg, J2 = 0.0 deg
};
P[212] {
   GP1:
       UF : 5, UT : 6,     CONFIG: 'N U T, 0, 0, 0',
      X = -157.0 mm, Y = -134.0 mm, Z = 85.8 mm,
      W = 0.0 deg, P = 0.0 deg, R = 0.0 deg
   GP2:
       UF : 1, UT : 2,
      J1 = 0.0 deg, J2 = 0.0 deg
};
P[213] {
   GP1:
       UF : 5, UT : 6,     CONFIG: 'N U T, 0, 0, 0',
      X = -150.0 mm, Y = -140.0 mm, Z = 85.8 mm,
      W = 0.0 deg, P = 0.0 deg, R = 0.0 deg
   GP2:
       UF : 1, UT : 2,
      J1 = 0.0 deg, J2 = 0.0 deg
};
P[214] {
   GP1:
       UF : 5, UT : 6,     CONFIG: 'N U T, 0, 0, 0',
      X = -155.0 mm, Y = -140.0 mm, Z = 85.8 mm,
      W = 0.0 deg, P = 0.0 deg, R = 0.0 deg
   GP2:
       UF : 1, UT : 2,
      J1 = 0.0 deg, J2 = 0.0 deg
};
P[215] {
   GP1:
       UF : 5, UT : 6,     CONFIG: 'N U T, 0, 0, 0',
      X = -157.0 mm, Y = -139.0 mm, Z = 85.8 mm,
      W = 0.0 deg, P = 0.0 deg, R = 0.0 deg
   GP2:
       UF : 1, UT : 2,
      J1 = 0.0 deg, J2 = 0.0 deg
};
P[216] {
   GP1:
       UF : 5, UT : 6,     CONFIG: 'N U T, 0, 0, 0',
      X = -157.0 mm, Y = -139.0 mm, Z = 89.1 mm,
      W = 0.0 deg, P = 0.0 deg, R = 0.0 deg
   GP2:
       UF : 1, UT : 2,
      J1 = 0.0 deg, J2 = 0.0 deg
};
P[217] {
   GP1:
       UF : 5, UT : 6,     CONFIG: 'N U T, 0, 0, 0',
      X = -113.0 mm, Y = -63.1 mm, Z = 89.1 mm,
      W = 0.0 deg, P = 0.0 deg, R = 0.0 deg
   GP2:
       UF : 1, UT : 2,
      J1 = 0.0 deg, J2 = 0.0 deg
};
P[218] {
   GP1:
       UF : 5, UT : 6,     CONFIG: 'N U T, 0, 0, 0',
      X = -112.0 mm, Y = -62.9 mm, Z = 89.1 mm,
      W = 0.0 deg, P = 0.0 deg, R = 0.0 deg
   GP2:
       UF : 1, UT : 2,
      J1 = 0.0 deg, J2 = 0.0 deg
};
P[219] {
   GP1:
       UF : 5, UT : 6,     CONFIG: 'N U T, 0, 0, 0',
      X = -111.0 mm, Y = -62.7 mm, Z = 89.1 mm,
      W = 0.0 deg, P = 0.0 deg, R = 0.0 deg
   GP2:
       UF : 1, UT : 2,
      J1 = 0.0 deg, J2 = 0.0 deg
};
P[220] {
   GP1:
       UF : 5, UT : 6,     CONFIG: 'N U T, 0, 0, 0',
      X = -109.0 mm, Y = -62.8 mm, Z = 89.1 mm,
      W = 0.0 deg, P = 0.0 deg, R = 0.0 deg
   GP2:
       UF : 1, UT : 2,
      J1 = 0.0 deg, J2 = 0.0 deg
};
P[221] {
   GP1:
       UF : 5, UT : 6,     CONFIG: 'N U T, 0, 0, 0',
      X = -108.0 mm, Y = -63.0 mm, Z = 89.1 mm,
      W = 0.0 deg, P = 0.0 deg, R = 0.0 deg
   GP2:
       UF : 1, UT : 2,
      J1 = 0.0 deg, J2 = 0.0 deg
};
P[222] {
   GP1:
       UF : 5, UT : 6,     CONFIG: 'N U T, 0, 0, 0',
      X = -107.0 mm, Y = -63.4 mm, Z = 89.1 mm,
      W = 0.0 deg, P = 0.0 deg, R = 0.0 deg
   GP2:
       UF : 1, UT : 2,
      J1 = 0.0 deg, J2 = 0.0 deg
};
P[223] {
   GP1:
       UF : 5, UT : 6,     CONFIG: 'N U T, 0, 0, 0',
      X = -106.0 mm, Y = -63.9 mm, Z = 89.1 mm,
      W = 0.0 deg, P = 0.0 deg, R = 0.0 deg
   GP2:
       UF : 1, UT : 2,
      J1 = 0.0 deg, J2 = 0.0 deg
};
P[224] {
   GP1:
       UF : 5, UT : 6,     CONFIG: 'N U T, 0, 0, 0',
      X = -104.0 mm, Y = -64.6 mm, Z = 89.1 mm,
      W = 0.0 deg, P = 0.0 deg, R = 0.0 deg
   GP2:
       UF : 1, UT : 2,
      J1 = 0.0 deg, J2 = 0.0 deg
};
P[225] {
   GP1:
       UF : 5, UT : 6,     CONFIG: 'N U T, 0, 0, 0',
      X = -103.0 mm, Y = -65.5 mm, Z = 89.1 mm,
      W = 0.0 deg, P = 0.0 deg, R = 0.0 deg
   GP2:
       UF : 1, UT : 2,
      J1 = 0.0 deg, J2 = 0.0 deg
};
P[226] {
   GP1:
       UF : 5, UT : 6,     CONFIG: 'N U T, 0, 0, 0',
      X = -102.0 mm, Y = -66.4 mm, Z = 89.1 mm,
      W = 0.0 deg, P = 0.0 deg, R = 0.0 deg
   GP2:
       UF : 1, UT : 2,
      J1 = 0.0 deg, J2 = 0.0 deg
};
P[227] {
   GP1:
       UF : 5, UT : 6,     CONFIG: 'N U T, 0, 0, 0',
      X = -101.0 mm, Y = -67.5 mm, Z = 89.1 mm,
      W = 0.0 deg, P = 0.0 deg, R = 0.0 deg
   GP2:
       UF : 1, UT : 2,
      J1 = 0.0 deg, J2 = 0.0 deg
};
P[228] {
   GP1:
       UF : 5, UT : 6,     CONFIG: 'N U T, 0, 0, 0',
      X = -101.0 mm, Y = -68.7 mm, Z = 89.1 mm,
      W = 0.0 deg, P = 0.0 deg, R = 0.0 deg
   GP2:
       UF : 1, UT : 2,
      J1 = 0.0 deg, J2 = 0.0 deg
};
P[229] {
   GP1:
       UF : 5, UT : 6,     CONFIG: 'N U T, 0, 0, 0',
      X = -100.0 mm, Y = -69.9 mm, Z = 89.1 mm,
      W = 0.0 deg, P = 0.0 deg, R = 0.0 deg
   GP2:
       UF : 1, UT : 2,
      J1 = 0.0 deg, J2 = 0.0 deg
};
P[230] {
   GP1:
       UF : 5, UT : 6,     CONFIG: 'N U T, 0, 0, 0',
      X = -99.7 mm, Y = -71.2 mm, Z = 89.1 mm,
      W = 0.0 deg, P = 0.0 deg, R = 0.0 deg
   GP2:
       UF : 1, UT : 2,
      J1 = 0.0 deg, J2 = 0.0 deg
};
P[231] {
   GP1:
       UF : 5, UT : 6,     CONFIG: 'N U T, 0, 0, 0',
      X = -95.8 mm, Y = -86.0 mm, Z = 89.1 mm,
      W = 0.0 deg, P = 0.0 deg, R = 0.0 deg
   GP2:
       UF : 1, UT : 2,
      J1 = 0.0 deg, J2 = 0.0 deg
};
P[232] {
   GP1:
       UF : 5, UT : 6,     CONFIG: 'N U T, 0, 0, 0',
      X = -95.5 mm, Y = -87.3 mm, Z = 89.1 mm,
      W = 0.0 deg, P = 0.0 deg, R = 0.0 deg
   GP2:
       UF : 1, UT : 2,
      J1 = 0.0 deg, J2 = 0.0 deg
};
P[233] {
   GP1:
       UF : 5, UT : 6,     CONFIG: 'N U T, 0, 0, 0',
      X = -95.4 mm, Y = -88.7 mm, Z = 89.1 mm,
      W = 0.0 deg, P = 0.0 deg, R = 0.0 deg
   GP2:
       UF : 1, UT : 2,
      J1 = 0.0 deg, J2 = 0.0 deg
};
P[234] {
   GP1:
       UF : 5, UT : 6,     CONFIG: 'N U T, 0, 0, 0',
      X = -95.5 mm, Y = -90.1 mm, Z = 89.1 mm,
      W = 0.0 deg, P = 0.0 deg, R = 0.0 deg
   GP2:
       UF : 1, UT : 2,
      J1 = 0.0 deg, J2 = 0.0 deg
};
P[235] {
   GP1:
       UF : 5, UT : 6,     CONFIG: 'N U T, 0, 0, 0',
      X = -95.7 mm, Y = -91.4 mm, Z = 89.1 mm,
      W = 0.0 deg, P = 0.0 deg, R = 0.0 deg
   GP2:
       UF : 1, UT : 2,
      J1 = 0.0 deg, J2 = 0.0 deg
};
P[236] {
   GP1:
       UF : 5, UT : 6,     CONFIG: 'N U T, 0, 0, 0',
      X = -96.1 mm, Y = -92.8 mm, Z = 89.1 mm,
      W = 0.0 deg, P = 0.0 deg, R = 0.0 deg
   GP2:
       UF : 1, UT : 2,
      J1 = 0.0 deg, J2 = 0.0 deg
};
P[237] {
   GP1:
       UF : 5, UT : 6,     CONFIG: 'N U T, 0, 0, 0',
      X = -96.6 mm, Y = -94.1 mm, Z = 89.1 mm,
      W = 0.0 deg, P = 0.0 deg, R = 0.0 deg
   GP2:
       UF : 1, UT : 2,
      J1 = 0.0 deg, J2 = 0.0 deg
};
P[238] {
   GP1:
       UF : 5, UT : 6,     CONFIG: 'N U T, 0, 0, 0',
      X = -97.3 mm, Y = -95.3 mm, Z = 89.1 mm,
      W = 0.0 deg, P = 0.0 deg, R = 0.0 deg
   GP2:
       UF : 1, UT : 2,
      J1 = 0.0 deg, J2 = 0.0 deg
};
P[239] {
   GP1:
